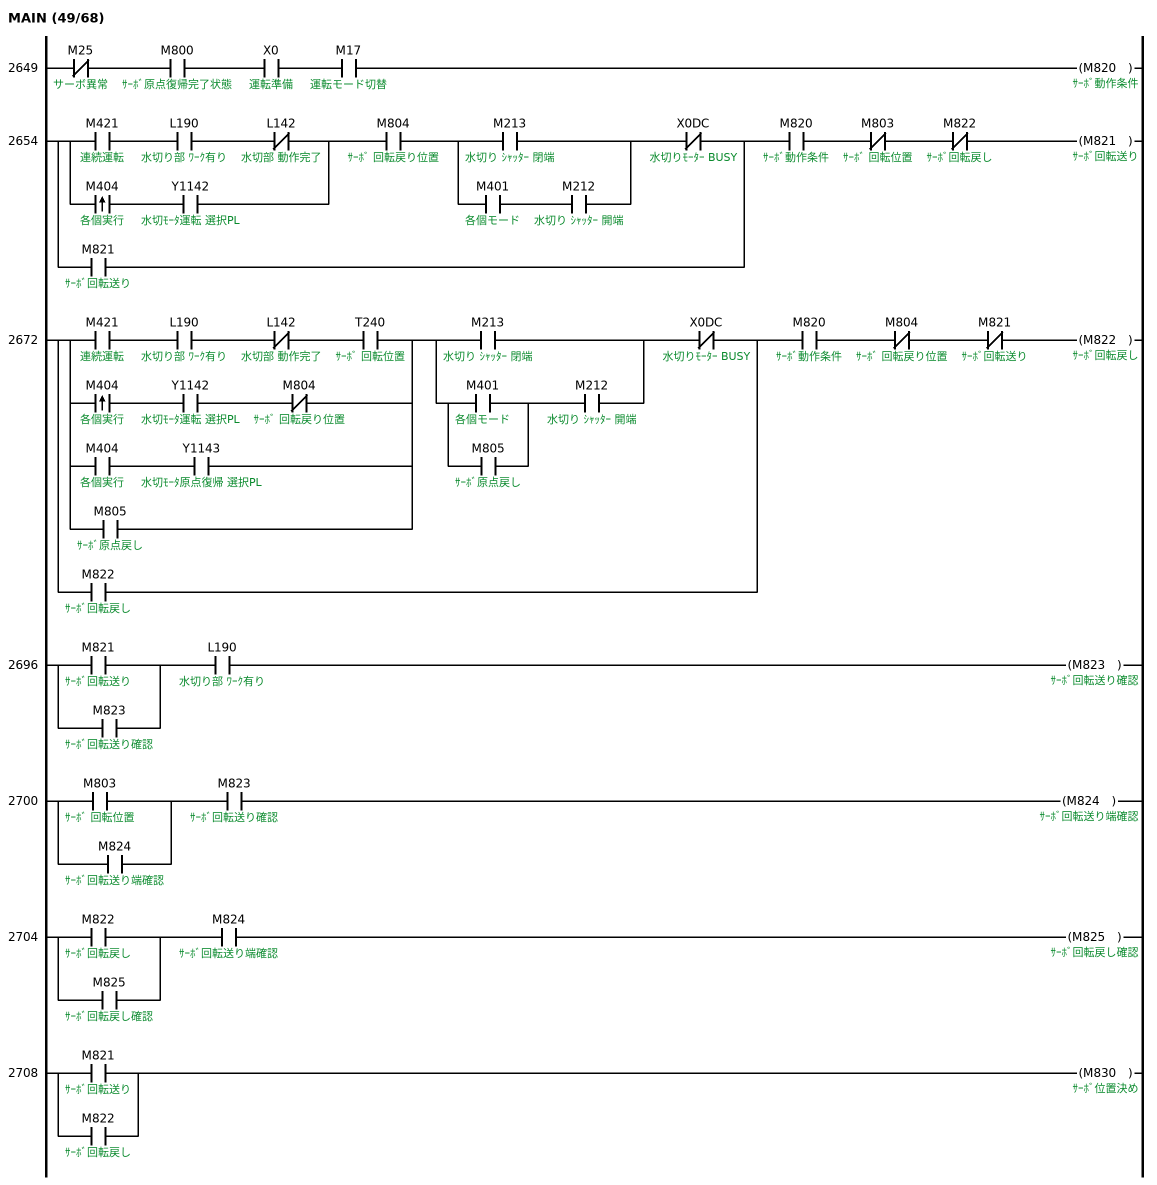
[picture p48: ladder of MAIN, rungs at steps 2649 to 2708]
2649  LDI     M25  ; サーボ異常
      AND     M800  ; ｻｰﾎﾞ原点復帰完了状態
      AND     X0  ; 運転準備
      AND     M17  ; 運転モード切替
      OUT     M820  ; ｻｰﾎﾞ動作条件
2654  LD      M421  ; 連続運転
      AND     L190  ; 水切り部 ﾜｰｸ有り
      ANI     L142  ; 水切部 動作完了
      LDP     M404  ; 各個実行
      AND     Y1142  ; 水切ﾓｰﾀ運転 選択PL
      ORB
      AND     M804  ; ｻｰﾎﾞ 回転戻り位置
      LD      M213  ; 水切り ｼｬｯﾀｰ 閉端
      LD      M401  ; 各個モード
      AND     M212  ; 水切り ｼｬｯﾀｰ 開端
      ORB
      ANB
      ANI     X0DC  ; 水切りﾓｰﾀｰ BUSY
      OR      M821  ; ｻｰﾎﾞ回転送り
      AND     M820  ; ｻｰﾎﾞ動作条件
      ANI     M803  ; ｻｰﾎﾞ 回転位置
      ANI     M822  ; ｻｰﾎﾞ回転戻し
      OUT     M821  ; ｻｰﾎﾞ回転送り
2672  LD      M421  ; 連続運転
      AND     L190  ; 水切り部 ﾜｰｸ有り
      ANI     L142  ; 水切部 動作完了
      AND     T240  ; ｻｰﾎﾞ 回転位置
      LDP     M404  ; 各個実行
      AND     Y1142  ; 水切ﾓｰﾀ運転 選択PL
      ANI     M804  ; ｻｰﾎﾞ 回転戻り位置
      ORB
      LD      M404  ; 各個実行
      AND     Y1143  ; 水切ﾓｰﾀ原点復帰 選択PL
      ORB
      OR      M805  ; ｻｰﾎﾞ原点戻し
      LD      M213  ; 水切り ｼｬｯﾀｰ 閉端
      LD      M401  ; 各個モード
      OR      M805  ; ｻｰﾎﾞ原点戻し
      AND     M212  ; 水切り ｼｬｯﾀｰ 開端
      ORB
      ANB
      ANI     X0DC  ; 水切りﾓｰﾀｰ BUSY
      OR      M822  ; ｻｰﾎﾞ回転戻し
      AND     M820  ; ｻｰﾎﾞ動作条件
      ANI     M804  ; ｻｰﾎﾞ 回転戻り位置
      ANI     M821  ; ｻｰﾎﾞ回転送り
      OUT     M822  ; ｻｰﾎﾞ回転戻し
2696  LD      M821  ; ｻｰﾎﾞ回転送り
      OR      M823  ; ｻｰﾎﾞ回転送り確認
      AND     L190  ; 水切り部 ﾜｰｸ有り
      OUT     M823  ; ｻｰﾎﾞ回転送り確認
2700  LD      M803  ; ｻｰﾎﾞ 回転位置
      OR      M824  ; ｻｰﾎﾞ回転送り端確認
      AND     M823  ; ｻｰﾎﾞ回転送り確認
      OUT     M824  ; ｻｰﾎﾞ回転送り端確認
2704  LD      M822  ; ｻｰﾎﾞ回転戻し
      OR      M825  ; ｻｰﾎﾞ回転戻し確認
      AND     M824  ; ｻｰﾎﾞ回転送り端確認
      OUT     M825  ; ｻｰﾎﾞ回転戻し確認
2708  LD      M821  ; ｻｰﾎﾞ回転送り
      OR      M822  ; ｻｰﾎﾞ回転戻し
      OUT     M830  ; ｻｰﾎﾞ位置決め
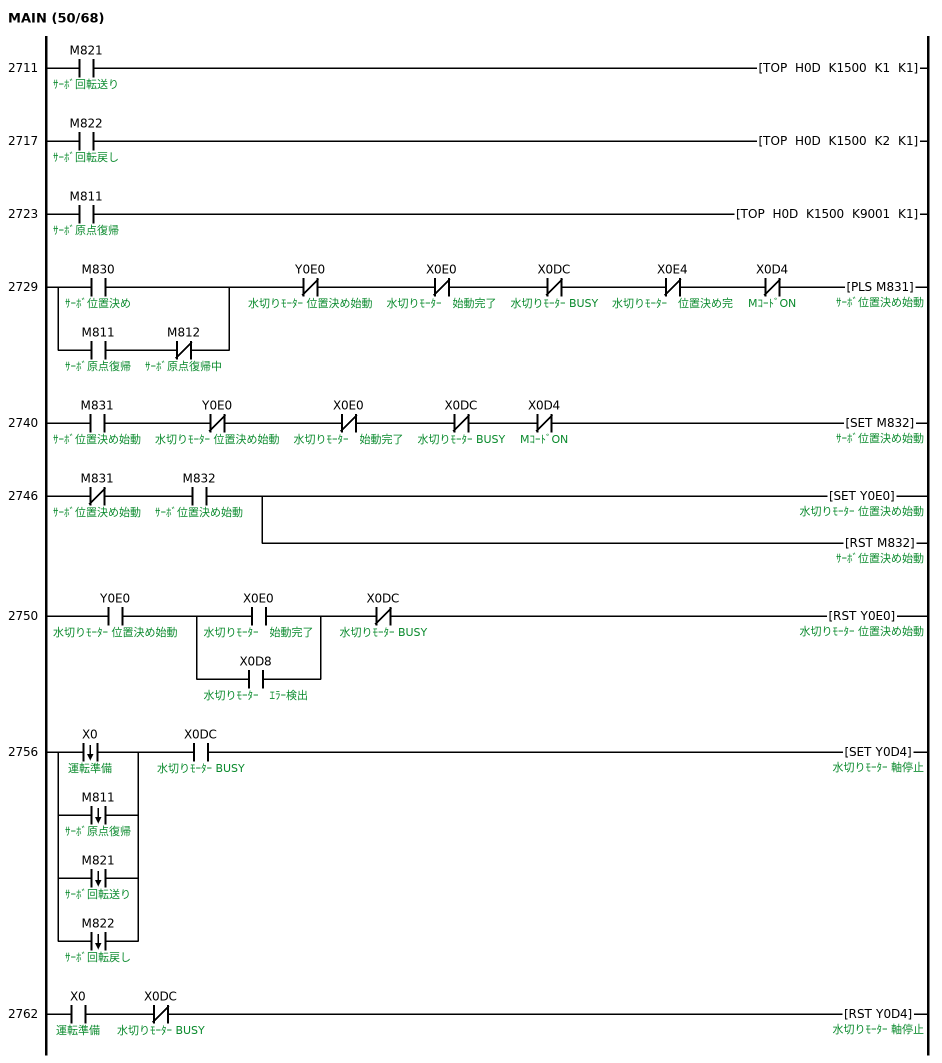
2711  LD      M821  ; ｻｰﾎﾞ回転送り
      TOP     H0D K1500 K1 K1
2717  LD      M822  ; ｻｰﾎﾞ回転戻し
      TOP     H0D K1500 K2 K1
2723  LD      M811  ; ｻｰﾎﾞ原点復帰
      TOP     H0D K1500 K9001 K1
2729  LD      M830  ; ｻｰﾎﾞ位置決め
      LD      M811  ; ｻｰﾎﾞ原点復帰
      ANI     M812  ; ｻｰﾎﾞ原点復帰中
      ORB
      ANI     Y0E0  ; 水切りﾓｰﾀｰ 位置決め始動
      ANI     X0E0  ; 水切りﾓｰﾀｰ　始動完了
      ANI     X0DC  ; 水切りﾓｰﾀｰ BUSY
      ANI     X0E4  ; 水切りﾓｰﾀｰ　位置決め完
      ANI     X0D4  ; MｺｰﾄﾞON
      PLS     M831  ; ｻｰﾎﾞ位置決め始動
2740  LD      M831  ; ｻｰﾎﾞ位置決め始動
      ANI     Y0E0  ; 水切りﾓｰﾀｰ 位置決め始動
      ANI     X0E0  ; 水切りﾓｰﾀｰ　始動完了
      ANI     X0DC  ; 水切りﾓｰﾀｰ BUSY
      ANI     X0D4  ; MｺｰﾄﾞON
      SET     M832  ; ｻｰﾎﾞ位置決め始動
2746  LDI     M831  ; ｻｰﾎﾞ位置決め始動
      AND     M832  ; ｻｰﾎﾞ位置決め始動
      SET     Y0E0  ; 水切りﾓｰﾀｰ 位置決め始動
      RST     M832  ; ｻｰﾎﾞ位置決め始動
2750  LD      Y0E0  ; 水切りﾓｰﾀｰ 位置決め始動
      LD      X0E0  ; 水切りﾓｰﾀｰ　始動完了
      OR      X0D8  ; 水切りﾓｰﾀｰ　ｴﾗｰ検出
      ANB
      ANI     X0DC  ; 水切りﾓｰﾀｰ BUSY
      RST     Y0E0  ; 水切りﾓｰﾀｰ 位置決め始動
2756  LDF     X0  ; 運転準備
      ORF     M811  ; ｻｰﾎﾞ原点復帰
      ORF     M821  ; ｻｰﾎﾞ回転送り
      ORF     M822  ; ｻｰﾎﾞ回転戻し
      AND     X0DC  ; 水切りﾓｰﾀｰ BUSY
      SET     Y0D4  ; 水切りﾓｰﾀｰ 軸停止
2762  LD      X0  ; 運転準備
      ANI     X0DC  ; 水切りﾓｰﾀｰ BUSY
      RST     Y0D4  ; 水切りﾓｰﾀｰ 軸停止
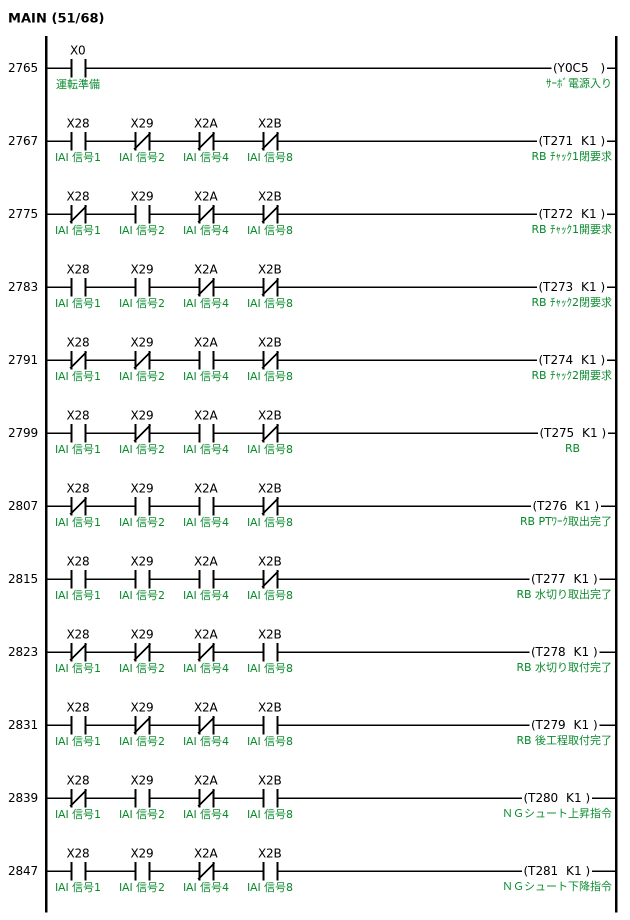
2765  LD      X0  ; 運転準備
      OUT     Y0C5  ; ｻｰﾎﾞ電源入り
2767  LD      X28  ; IAI 信号1
      ANI     X29  ; IAI 信号2
      ANI     X2A  ; IAI 信号4
      ANI     X2B  ; IAI 信号8
      OUT     T271 K1  ; RB ﾁｬｯｸ1閉要求
2775  LDI     X28  ; IAI 信号1
      AND     X29  ; IAI 信号2
      ANI     X2A  ; IAI 信号4
      ANI     X2B  ; IAI 信号8
      OUT     T272 K1  ; RB ﾁｬｯｸ1開要求
2783  LD      X28  ; IAI 信号1
      AND     X29  ; IAI 信号2
      ANI     X2A  ; IAI 信号4
      ANI     X2B  ; IAI 信号8
      OUT     T273 K1  ; RB ﾁｬｯｸ2閉要求
2791  LDI     X28  ; IAI 信号1
      ANI     X29  ; IAI 信号2
      AND     X2A  ; IAI 信号4
      ANI     X2B  ; IAI 信号8
      OUT     T274 K1  ; RB ﾁｬｯｸ2開要求
2799  LD      X28  ; IAI 信号1
      ANI     X29  ; IAI 信号2
      AND     X2A  ; IAI 信号4
      ANI     X2B  ; IAI 信号8
      OUT     T275 K1  ; RB
2807  LDI     X28  ; IAI 信号1
      AND     X29  ; IAI 信号2
      AND     X2A  ; IAI 信号4
      ANI     X2B  ; IAI 信号8
      OUT     T276 K1  ; RB PTﾜｰｸ取出完了
2815  LD      X28  ; IAI 信号1
      AND     X29  ; IAI 信号2
      AND     X2A  ; IAI 信号4
      ANI     X2B  ; IAI 信号8
      OUT     T277 K1  ; RB 水切り取出完了
2823  LDI     X28  ; IAI 信号1
      ANI     X29  ; IAI 信号2
      ANI     X2A  ; IAI 信号4
      AND     X2B  ; IAI 信号8
      OUT     T278 K1  ; RB 水切り取付完了
2831  LD      X28  ; IAI 信号1
      ANI     X29  ; IAI 信号2
      ANI     X2A  ; IAI 信号4
      AND     X2B  ; IAI 信号8
      OUT     T279 K1  ; RB 後工程取付完了
2839  LDI     X28  ; IAI 信号1
      AND     X29  ; IAI 信号2
      ANI     X2A  ; IAI 信号4
      AND     X2B  ; IAI 信号8
      OUT     T280 K1  ; ＮＧシュート上昇指令
2847  LD      X28  ; IAI 信号1
      AND     X29  ; IAI 信号2
      ANI     X2A  ; IAI 信号4
      AND     X2B  ; IAI 信号8
      OUT     T281 K1  ; ＮＧシュート下降指令
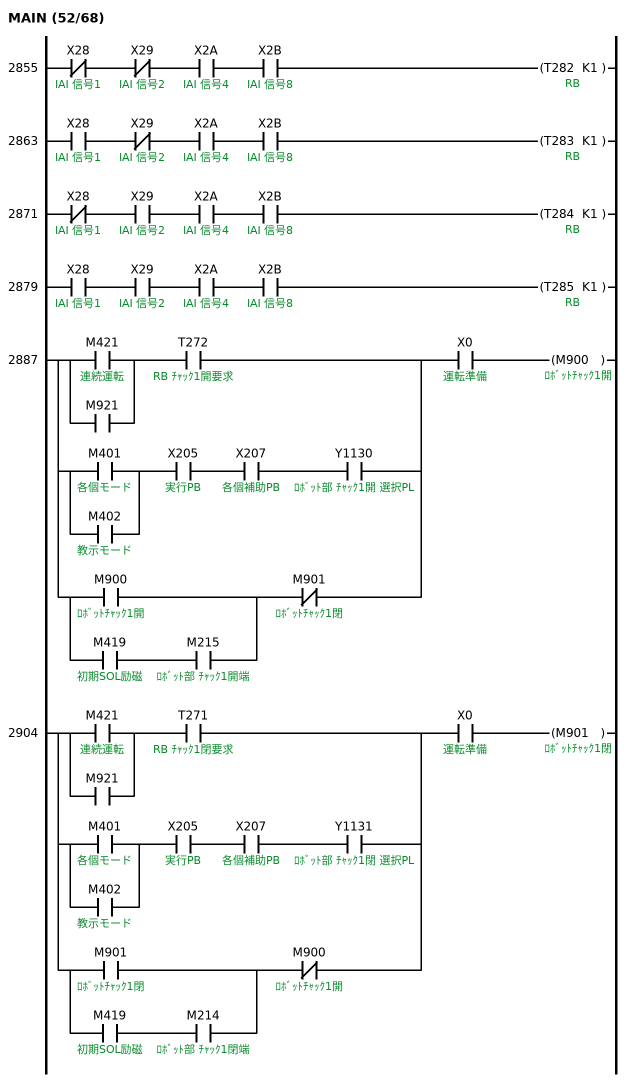
2855  LDI     X28  ; IAI 信号1
      ANI     X29  ; IAI 信号2
      AND     X2A  ; IAI 信号4
      AND     X2B  ; IAI 信号8
      OUT     T282 K1  ; RB
2863  LD      X28  ; IAI 信号1
      ANI     X29  ; IAI 信号2
      AND     X2A  ; IAI 信号4
      AND     X2B  ; IAI 信号8
      OUT     T283 K1  ; RB
2871  LDI     X28  ; IAI 信号1
      AND     X29  ; IAI 信号2
      AND     X2A  ; IAI 信号4
      AND     X2B  ; IAI 信号8
      OUT     T284 K1  ; RB
2879  LD      X28  ; IAI 信号1
      AND     X29  ; IAI 信号2
      AND     X2A  ; IAI 信号4
      AND     X2B  ; IAI 信号8
      OUT     T285 K1  ; RB
2887  LD      M421  ; 連続運転
      OR      M921
      AND     T272  ; RB ﾁｬｯｸ1開要求
      LD      M401  ; 各個モード
      OR      M402  ; 教示モード
      AND     X205  ; 実行PB
      AND     X207  ; 各個補助PB
      AND     Y1130  ; ﾛﾎﾞｯﾄ部 ﾁｬｯｸ1開 選択PL
      ORB
      LD      M900  ; ﾛﾎﾞｯﾄﾁｬｯｸ1開
      LD      M419  ; 初期SOL励磁
      AND     M215  ; ﾛﾎﾞｯﾄ部 ﾁｬｯｸ1開端
      ORB
      ANI     M901  ; ﾛﾎﾞｯﾄﾁｬｯｸ1閉
      ORB
      AND     X0  ; 運転準備
      OUT     M900  ; ﾛﾎﾞｯﾄﾁｬｯｸ1開
2904  LD      M421  ; 連続運転
      OR      M921
      AND     T271  ; RB ﾁｬｯｸ1閉要求
      LD      M401  ; 各個モード
      OR      M402  ; 教示モード
      AND     X205  ; 実行PB
      AND     X207  ; 各個補助PB
      AND     Y1131  ; ﾛﾎﾞｯﾄ部 ﾁｬｯｸ1閉 選択PL
      ORB
      LD      M901  ; ﾛﾎﾞｯﾄﾁｬｯｸ1閉
      LD      M419  ; 初期SOL励磁
      AND     M214  ; ﾛﾎﾞｯﾄ部 ﾁｬｯｸ1閉端
      ORB
      ANI     M900  ; ﾛﾎﾞｯﾄﾁｬｯｸ1開
      ORB
      AND     X0  ; 運転準備
      OUT     M901  ; ﾛﾎﾞｯﾄﾁｬｯｸ1閉
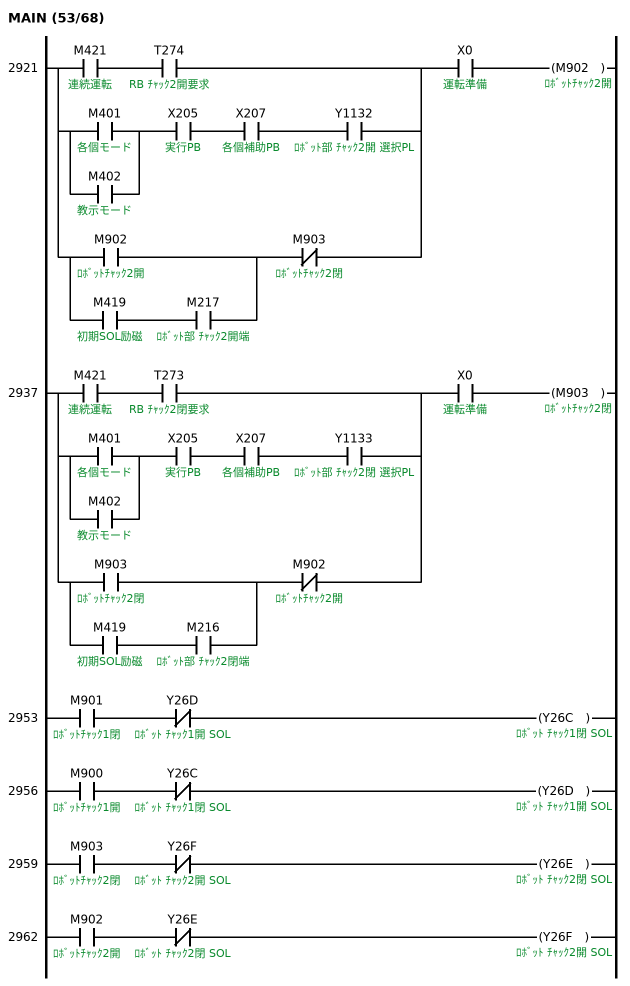
2921  LD      M421  ; 連続運転
      AND     T274  ; RB ﾁｬｯｸ2開要求
      LD      M401  ; 各個モード
      OR      M402  ; 教示モード
      AND     X205  ; 実行PB
      AND     X207  ; 各個補助PB
      AND     Y1132  ; ﾛﾎﾞｯﾄ部 ﾁｬｯｸ2開 選択PL
      ORB
      LD      M902  ; ﾛﾎﾞｯﾄﾁｬｯｸ2開
      LD      M419  ; 初期SOL励磁
      AND     M217  ; ﾛﾎﾞｯﾄ部 ﾁｬｯｸ2開端
      ORB
      ANI     M903  ; ﾛﾎﾞｯﾄﾁｬｯｸ2閉
      ORB
      AND     X0  ; 運転準備
      OUT     M902  ; ﾛﾎﾞｯﾄﾁｬｯｸ2開
2937  LD      M421  ; 連続運転
      AND     T273  ; RB ﾁｬｯｸ2閉要求
      LD      M401  ; 各個モード
      OR      M402  ; 教示モード
      AND     X205  ; 実行PB
      AND     X207  ; 各個補助PB
      AND     Y1133  ; ﾛﾎﾞｯﾄ部 ﾁｬｯｸ2閉 選択PL
      ORB
      LD      M903  ; ﾛﾎﾞｯﾄﾁｬｯｸ2閉
      LD      M419  ; 初期SOL励磁
      AND     M216  ; ﾛﾎﾞｯﾄ部 ﾁｬｯｸ2閉端
      ORB
      ANI     M902  ; ﾛﾎﾞｯﾄﾁｬｯｸ2開
      ORB
      AND     X0  ; 運転準備
      OUT     M903  ; ﾛﾎﾞｯﾄﾁｬｯｸ2閉
2953  LD      M901  ; ﾛﾎﾞｯﾄﾁｬｯｸ1閉
      ANI     Y26D  ; ﾛﾎﾞｯﾄ ﾁｬｯｸ1開 SOL
      OUT     Y26C  ; ﾛﾎﾞｯﾄ ﾁｬｯｸ1閉 SOL
2956  LD      M900  ; ﾛﾎﾞｯﾄﾁｬｯｸ1開
      ANI     Y26C  ; ﾛﾎﾞｯﾄ ﾁｬｯｸ1閉 SOL
      OUT     Y26D  ; ﾛﾎﾞｯﾄ ﾁｬｯｸ1開 SOL
2959  LD      M903  ; ﾛﾎﾞｯﾄﾁｬｯｸ2閉
      ANI     Y26F  ; ﾛﾎﾞｯﾄ ﾁｬｯｸ2開 SOL
      OUT     Y26E  ; ﾛﾎﾞｯﾄ ﾁｬｯｸ2閉 SOL
2962  LD      M902  ; ﾛﾎﾞｯﾄﾁｬｯｸ2開
      ANI     Y26E  ; ﾛﾎﾞｯﾄ ﾁｬｯｸ2閉 SOL
      OUT     Y26F  ; ﾛﾎﾞｯﾄ ﾁｬｯｸ2開 SOL
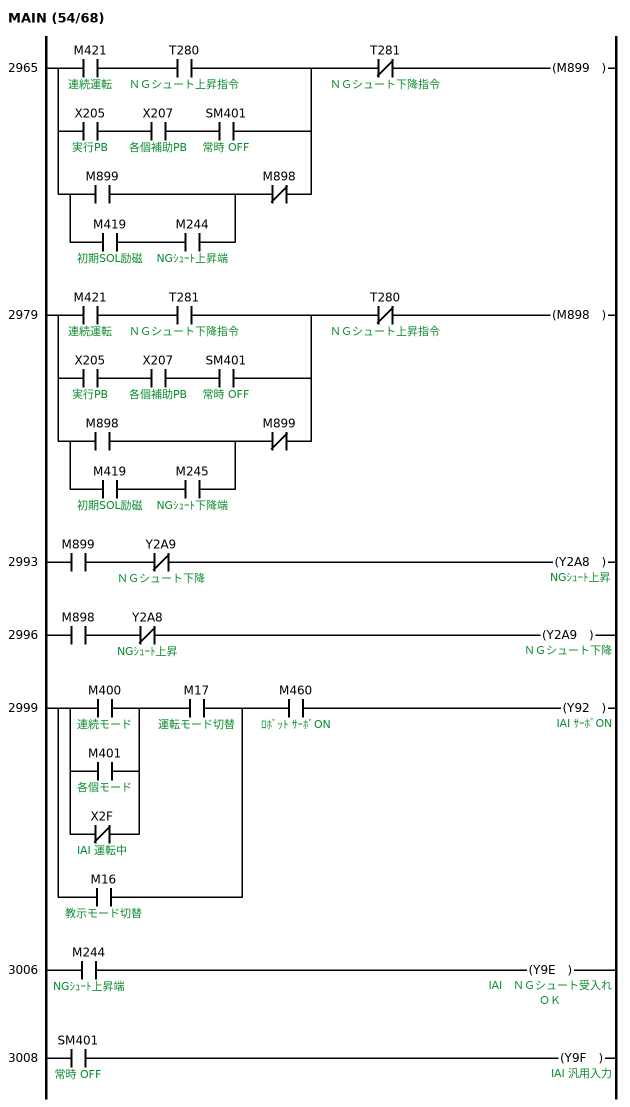
2965  LD      M421  ; 連続運転
      AND     T280  ; ＮＧシュート上昇指令
      LD      X205  ; 実行PB
      AND     X207  ; 各個補助PB
      AND     SM401  ; 常時 OFF
      ORB
      LD      M899
      LD      M419  ; 初期SOL励磁
      AND     M244  ; NGｼｭｰﾄ上昇端
      ORB
      ANI     M898
      ORB
      ANI     T281  ; ＮＧシュート下降指令
      OUT     M899
2979  LD      M421  ; 連続運転
      AND     T281  ; ＮＧシュート下降指令
      LD      X205  ; 実行PB
      AND     X207  ; 各個補助PB
      AND     SM401  ; 常時 OFF
      ORB
      LD      M898
      LD      M419  ; 初期SOL励磁
      AND     M245  ; NGｼｭｰﾄ下降端
      ORB
      ANI     M899
      ORB
      ANI     T280  ; ＮＧシュート上昇指令
      OUT     M898
2993  LD      M899
      ANI     Y2A9  ; ＮＧシュート下降
      OUT     Y2A8  ; NGｼｭｰﾄ上昇
2996  LD      M898
      ANI     Y2A8  ; NGｼｭｰﾄ上昇
      OUT     Y2A9  ; ＮＧシュート下降
2999  LD      M400  ; 連続モード
      OR      M401  ; 各個モード
      ORI     X2F  ; IAI 運転中
      AND     M17  ; 運転モード切替
      OR      M16  ; 教示モード切替
      AND     M460  ; ﾛﾎﾞｯﾄ ｻｰﾎﾞON
      OUT     Y92  ; IAI ｻｰﾎﾞON
3006  LD      M244  ; NGｼｭｰﾄ上昇端
      OUT     Y9E  ; IAI　ＮＧシュート受入れＯＫ
3008  LD      SM401  ; 常時 OFF
      OUT     Y9F  ; IAI 汎用入力
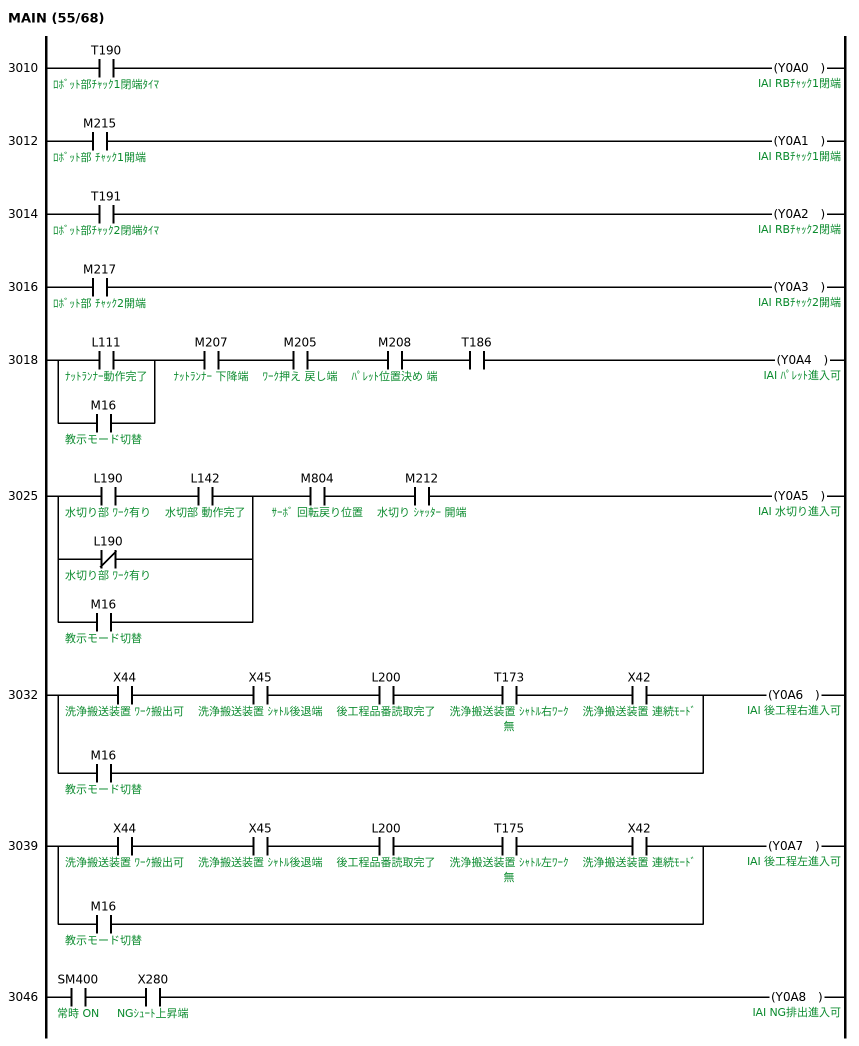
3010  LD      T190  ; ﾛﾎﾞｯﾄ部ﾁｬｯｸ1閉端ﾀｲﾏ
      OUT     Y0A0  ; IAI RBﾁｬｯｸ1閉端
3012  LD      M215  ; ﾛﾎﾞｯﾄ部 ﾁｬｯｸ1開端
      OUT     Y0A1  ; IAI RBﾁｬｯｸ1開端
3014  LD      T191  ; ﾛﾎﾞｯﾄ部ﾁｬｯｸ2閉端ﾀｲﾏ
      OUT     Y0A2  ; IAI RBﾁｬｯｸ2閉端
3016  LD      M217  ; ﾛﾎﾞｯﾄ部 ﾁｬｯｸ2開端
      OUT     Y0A3  ; IAI RBﾁｬｯｸ2開端
3018  LD      L111  ; ﾅｯﾄﾗﾝﾅｰ動作完了
      OR      M16  ; 教示モード切替
      AND     M207  ; ﾅｯﾄﾗﾝﾅｰ 下降端
      AND     M205  ; ﾜｰｸ押え 戻し端
      AND     M208  ; ﾊﾟﾚｯﾄ位置決め 端
      AND     T186
      OUT     Y0A4  ; IAI ﾊﾟﾚｯﾄ進入可
3025  LD      L190  ; 水切り部 ﾜｰｸ有り
      AND     L142  ; 水切部 動作完了
      ORI     L190  ; 水切り部 ﾜｰｸ有り
      OR      M16  ; 教示モード切替
      AND     M804  ; ｻｰﾎﾞ 回転戻り位置
      AND     M212  ; 水切り ｼｬｯﾀｰ 開端
      OUT     Y0A5  ; IAI 水切り進入可
3032  LD      X44  ; 洗浄搬送装置 ﾜｰｸ搬出可
      AND     X45  ; 洗浄搬送装置 ｼｬﾄﾙ後退端
      AND     L200  ; 後工程品番読取完了
      AND     T173  ; 洗浄搬送装置 ｼｬﾄﾙ右ﾜｰｸ無
      AND     X42  ; 洗浄搬送装置 連続ﾓｰﾄﾞ
      OR      M16  ; 教示モード切替
      OUT     Y0A6  ; IAI 後工程右進入可
3039  LD      X44  ; 洗浄搬送装置 ﾜｰｸ搬出可
      AND     X45  ; 洗浄搬送装置 ｼｬﾄﾙ後退端
      AND     L200  ; 後工程品番読取完了
      AND     T175  ; 洗浄搬送装置 ｼｬﾄﾙ左ﾜｰｸ無
      AND     X42  ; 洗浄搬送装置 連続ﾓｰﾄﾞ
      OR      M16  ; 教示モード切替
      OUT     Y0A7  ; IAI 後工程左進入可
3046  LD      SM400  ; 常時 ON
      AND     X280  ; NGｼｭｰﾄ上昇端
      OUT     Y0A8  ; IAI NG排出進入可
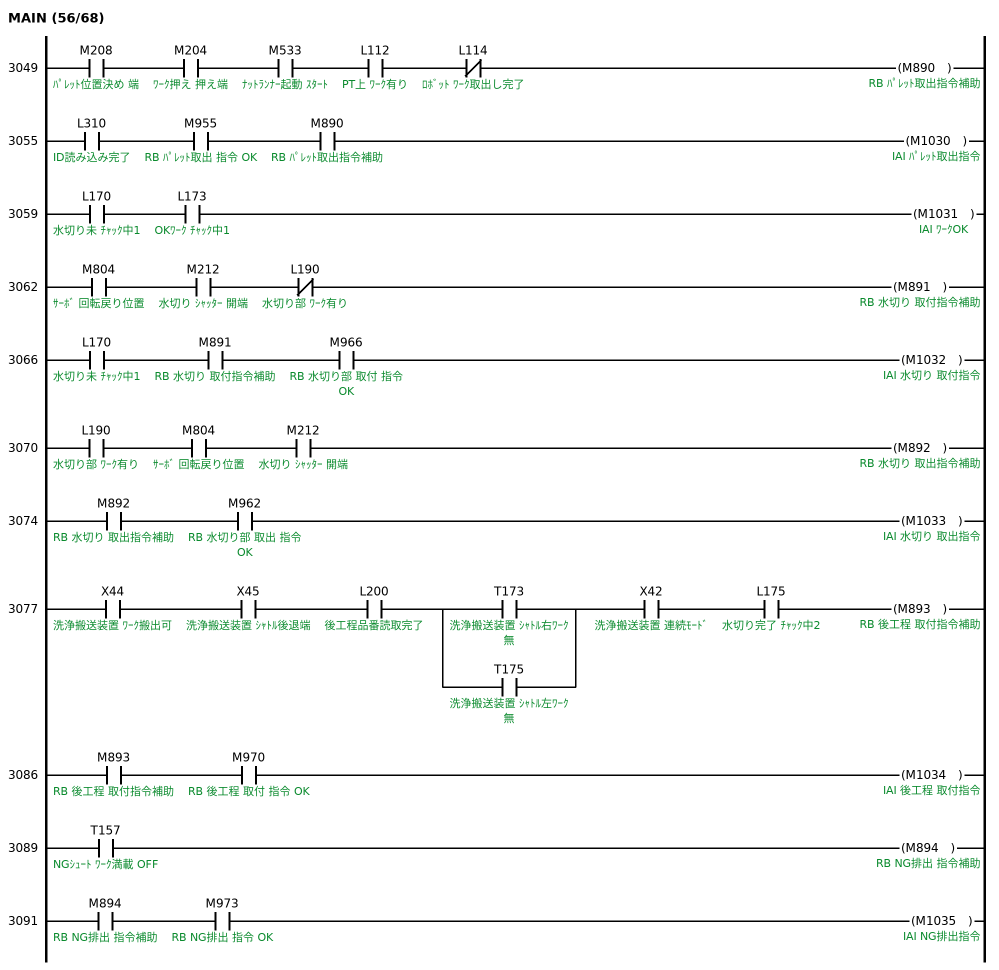
3049  LD      M208  ; ﾊﾟﾚｯﾄ位置決め 端
      AND     M204  ; ﾜｰｸ押え 押え端
      AND     M533  ; ﾅｯﾄﾗﾝﾅｰ起動 ｽﾀｰﾄ
      AND     L112  ; PT上 ﾜｰｸ有り
      ANI     L114  ; ﾛﾎﾞｯﾄ ﾜｰｸ取出し完了
      OUT     M890  ; RB ﾊﾟﾚｯﾄ取出指令補助
3055  LD      L310  ; ID読み込み完了
      AND     M955  ; RB ﾊﾟﾚｯﾄ取出 指令 OK
      AND     M890  ; RB ﾊﾟﾚｯﾄ取出指令補助
      OUT     M1030  ; IAI ﾊﾟﾚｯﾄ取出指令
3059  LD      L170  ; 水切り未 ﾁｬｯｸ中1
      AND     L173  ; OKﾜｰｸ ﾁｬｯｸ中1
      OUT     M1031  ; IAI ﾜｰｸOK
3062  LD      M804  ; ｻｰﾎﾞ 回転戻り位置
      AND     M212  ; 水切り ｼｬｯﾀｰ 開端
      ANI     L190  ; 水切り部 ﾜｰｸ有り
      OUT     M891  ; RB 水切り 取付指令補助
3066  LD      L170  ; 水切り未 ﾁｬｯｸ中1
      AND     M891  ; RB 水切り 取付指令補助
      AND     M966  ; RB 水切り部 取付 指令 OK
      OUT     M1032  ; IAI 水切り 取付指令
3070  LD      L190  ; 水切り部 ﾜｰｸ有り
      AND     M804  ; ｻｰﾎﾞ 回転戻り位置
      AND     M212  ; 水切り ｼｬｯﾀｰ 開端
      OUT     M892  ; RB 水切り 取出指令補助
3074  LD      M892  ; RB 水切り 取出指令補助
      AND     M962  ; RB 水切り部 取出 指令 OK
      OUT     M1033  ; IAI 水切り 取出指令
3077  LD      X44  ; 洗浄搬送装置 ﾜｰｸ搬出可
      AND     X45  ; 洗浄搬送装置 ｼｬﾄﾙ後退端
      AND     L200  ; 後工程品番読取完了
      LD      T173  ; 洗浄搬送装置 ｼｬﾄﾙ右ﾜｰｸ無
      OR      T175  ; 洗浄搬送装置 ｼｬﾄﾙ左ﾜｰｸ無
      ANB
      AND     X42  ; 洗浄搬送装置 連続ﾓｰﾄﾞ
      AND     L175  ; 水切り完了 ﾁｬｯｸ中2
      OUT     M893  ; RB 後工程 取付指令補助
3086  LD      M893  ; RB 後工程 取付指令補助
      AND     M970  ; RB 後工程 取付 指令 OK
      OUT     M1034  ; IAI 後工程 取付指令
3089  LD      T157  ; NGｼｭｰﾄ ﾜｰｸ満載 OFF
      OUT     M894  ; RB NG排出 指令補助
3091  LD      M894  ; RB NG排出 指令補助
      AND     M973  ; RB NG排出 指令 OK
      OUT     M1035  ; IAI NG排出指令
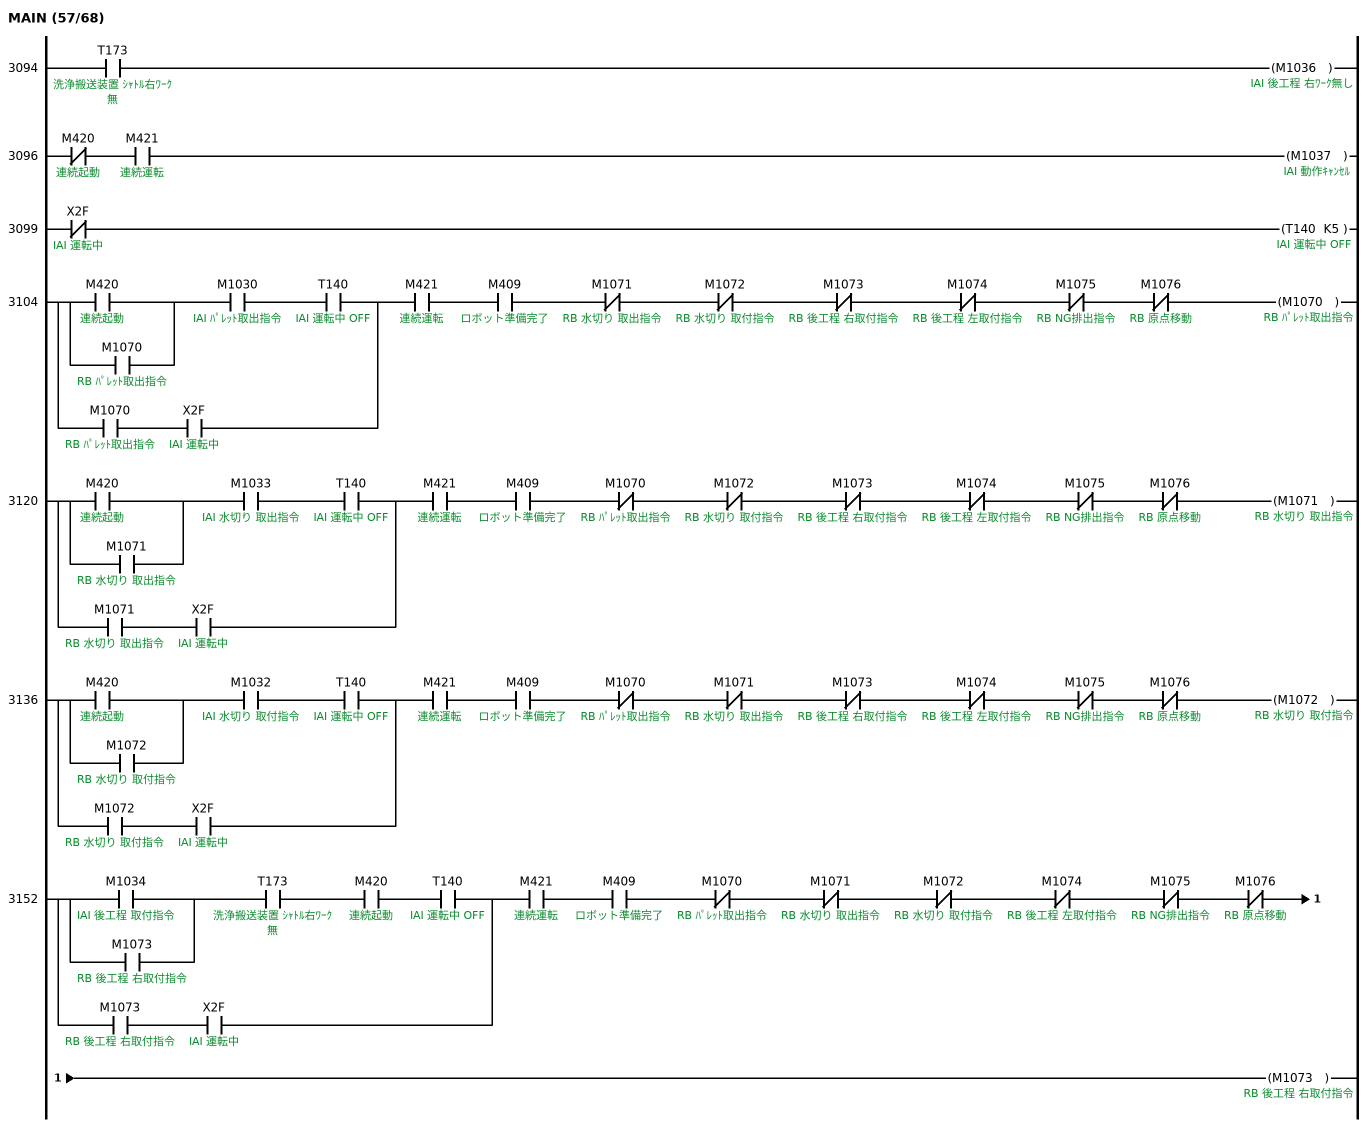
3094  LD      T173  ; 洗浄搬送装置 ｼｬﾄﾙ右ﾜｰｸ無
      OUT     M1036  ; IAI 後工程 右ﾜｰｸ無し
3096  LDI     M420  ; 連続起動
      AND     M421  ; 連続運転
      OUT     M1037  ; IAI 動作ｷｬﾝｾﾙ
3099  LDI     X2F  ; IAI 運転中
      OUT     T140 K5  ; IAI 運転中 OFF
3104  LD      M420  ; 連続起動
      OR      M1070  ; RB ﾊﾟﾚｯﾄ取出指令
      AND     M1030  ; IAI ﾊﾟﾚｯﾄ取出指令
      AND     T140  ; IAI 運転中 OFF
      LD      M1070  ; RB ﾊﾟﾚｯﾄ取出指令
      AND     X2F  ; IAI 運転中
      ORB
      AND     M421  ; 連続運転
      AND     M409  ; ロボット準備完了
      ANI     M1071  ; RB 水切り 取出指令
      ANI     M1072  ; RB 水切り 取付指令
      ANI     M1073  ; RB 後工程 右取付指令
      ANI     M1074  ; RB 後工程 左取付指令
      ANI     M1075  ; RB NG排出指令
      ANI     M1076  ; RB 原点移動
      OUT     M1070  ; RB ﾊﾟﾚｯﾄ取出指令
3120  LD      M420  ; 連続起動
      OR      M1071  ; RB 水切り 取出指令
      AND     M1033  ; IAI 水切り 取出指令
      AND     T140  ; IAI 運転中 OFF
      LD      M1071  ; RB 水切り 取出指令
      AND     X2F  ; IAI 運転中
      ORB
      AND     M421  ; 連続運転
      AND     M409  ; ロボット準備完了
      ANI     M1070  ; RB ﾊﾟﾚｯﾄ取出指令
      ANI     M1072  ; RB 水切り 取付指令
      ANI     M1073  ; RB 後工程 右取付指令
      ANI     M1074  ; RB 後工程 左取付指令
      ANI     M1075  ; RB NG排出指令
      ANI     M1076  ; RB 原点移動
      OUT     M1071  ; RB 水切り 取出指令
3136  LD      M420  ; 連続起動
      OR      M1072  ; RB 水切り 取付指令
      AND     M1032  ; IAI 水切り 取付指令
      AND     T140  ; IAI 運転中 OFF
      LD      M1072  ; RB 水切り 取付指令
      AND     X2F  ; IAI 運転中
      ORB
      AND     M421  ; 連続運転
      AND     M409  ; ロボット準備完了
      ANI     M1070  ; RB ﾊﾟﾚｯﾄ取出指令
      ANI     M1071  ; RB 水切り 取出指令
      ANI     M1073  ; RB 後工程 右取付指令
      ANI     M1074  ; RB 後工程 左取付指令
      ANI     M1075  ; RB NG排出指令
      ANI     M1076  ; RB 原点移動
      OUT     M1072  ; RB 水切り 取付指令
3152  LD      M1034  ; IAI 後工程 取付指令
      OR      M1073  ; RB 後工程 右取付指令
      AND     T173  ; 洗浄搬送装置 ｼｬﾄﾙ右ﾜｰｸ無
      AND     M420  ; 連続起動
      AND     T140  ; IAI 運転中 OFF
      LD      M1073  ; RB 後工程 右取付指令
      AND     X2F  ; IAI 運転中
      ORB
      AND     M421  ; 連続運転
      AND     M409  ; ロボット準備完了
      ANI     M1070  ; RB ﾊﾟﾚｯﾄ取出指令
      ANI     M1071  ; RB 水切り 取出指令
      ANI     M1072  ; RB 水切り 取付指令
      ANI     M1074  ; RB 後工程 左取付指令
      ANI     M1075  ; RB NG排出指令
      ANI     M1076  ; RB 原点移動
      OUT     M1073  ; RB 後工程 右取付指令
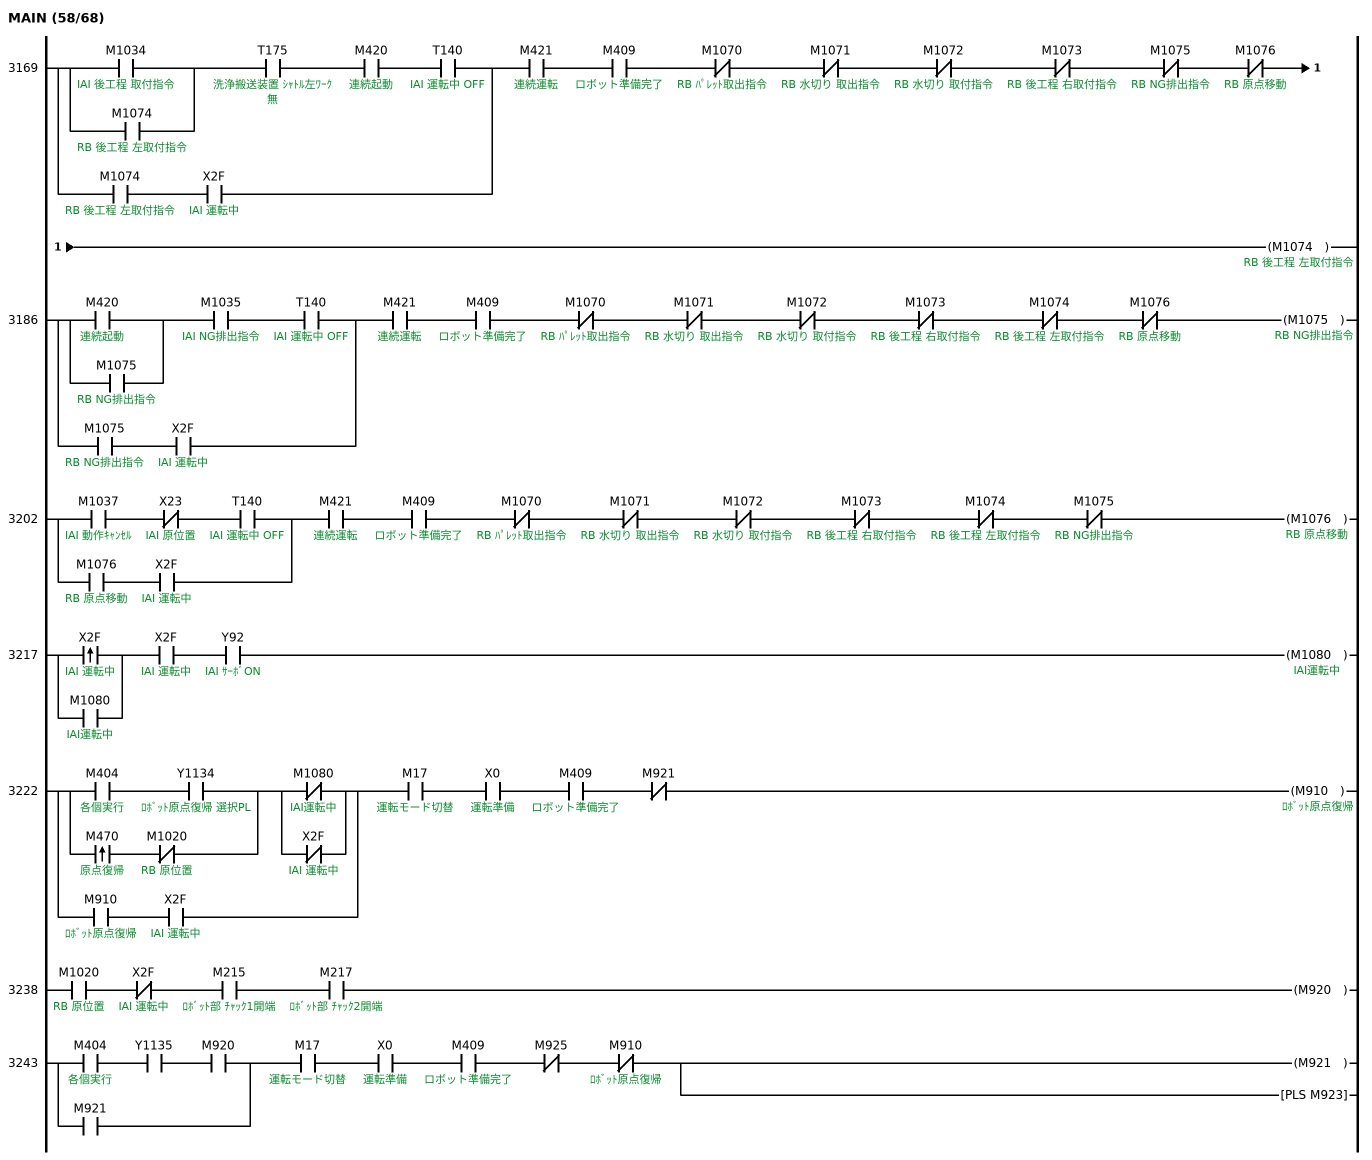
3169  LD      M1034  ; IAI 後工程 取付指令
      OR      M1074  ; RB 後工程 左取付指令
      AND     T175  ; 洗浄搬送装置 ｼｬﾄﾙ左ﾜｰｸ無
      AND     M420  ; 連続起動
      AND     T140  ; IAI 運転中 OFF
      LD      M1074  ; RB 後工程 左取付指令
      AND     X2F  ; IAI 運転中
      ORB
      AND     M421  ; 連続運転
      AND     M409  ; ロボット準備完了
      ANI     M1070  ; RB ﾊﾟﾚｯﾄ取出指令
      ANI     M1071  ; RB 水切り 取出指令
      ANI     M1072  ; RB 水切り 取付指令
      ANI     M1073  ; RB 後工程 右取付指令
      ANI     M1075  ; RB NG排出指令
      ANI     M1076  ; RB 原点移動
      OUT     M1074  ; RB 後工程 左取付指令
3186  LD      M420  ; 連続起動
      OR      M1075  ; RB NG排出指令
      AND     M1035  ; IAI NG排出指令
      AND     T140  ; IAI 運転中 OFF
      LD      M1075  ; RB NG排出指令
      AND     X2F  ; IAI 運転中
      ORB
      AND     M421  ; 連続運転
      AND     M409  ; ロボット準備完了
      ANI     M1070  ; RB ﾊﾟﾚｯﾄ取出指令
      ANI     M1071  ; RB 水切り 取出指令
      ANI     M1072  ; RB 水切り 取付指令
      ANI     M1073  ; RB 後工程 右取付指令
      ANI     M1074  ; RB 後工程 左取付指令
      ANI     M1076  ; RB 原点移動
      OUT     M1075  ; RB NG排出指令
3202  LD      M1037  ; IAI 動作ｷｬﾝｾﾙ
      ANI     X23  ; IAI 原位置
      AND     T140  ; IAI 運転中 OFF
      LD      M1076  ; RB 原点移動
      AND     X2F  ; IAI 運転中
      ORB
      AND     M421  ; 連続運転
      AND     M409  ; ロボット準備完了
      ANI     M1070  ; RB ﾊﾟﾚｯﾄ取出指令
      ANI     M1071  ; RB 水切り 取出指令
      ANI     M1072  ; RB 水切り 取付指令
      ANI     M1073  ; RB 後工程 右取付指令
      ANI     M1074  ; RB 後工程 左取付指令
      ANI     M1075  ; RB NG排出指令
      OUT     M1076  ; RB 原点移動
3217  LDP     X2F  ; IAI 運転中
      OR      M1080  ; IAI運転中
      AND     X2F  ; IAI 運転中
      AND     Y92  ; IAI ｻｰﾎﾞON
      OUT     M1080  ; IAI運転中
3222  LD      M404  ; 各個実行
      AND     Y1134  ; ﾛﾎﾞｯﾄ原点復帰 選択PL
      LDP     M470  ; 原点復帰
      ANI     M1020  ; RB 原位置
      ORB
      LDI     M1080  ; IAI運転中
      ORI     X2F  ; IAI 運転中
      ANB
      LD      M910  ; ﾛﾎﾞｯﾄ原点復帰
      AND     X2F  ; IAI 運転中
      ORB
      AND     M17  ; 運転モード切替
      AND     X0  ; 運転準備
      AND     M409  ; ロボット準備完了
      ANI     M921
      OUT     M910  ; ﾛﾎﾞｯﾄ原点復帰
3238  LD      M1020  ; RB 原位置
      ANI     X2F  ; IAI 運転中
      AND     M215  ; ﾛﾎﾞｯﾄ部 ﾁｬｯｸ1開端
      AND     M217  ; ﾛﾎﾞｯﾄ部 ﾁｬｯｸ2開端
      OUT     M920
3243  LD      M404  ; 各個実行
      AND     Y1135
      AND     M920
      OR      M921
      AND     M17  ; 運転モード切替
      AND     X0  ; 運転準備
      AND     M409  ; ロボット準備完了
      ANI     M925
      ANI     M910  ; ﾛﾎﾞｯﾄ原点復帰
      OUT     M921
      PLS     M923
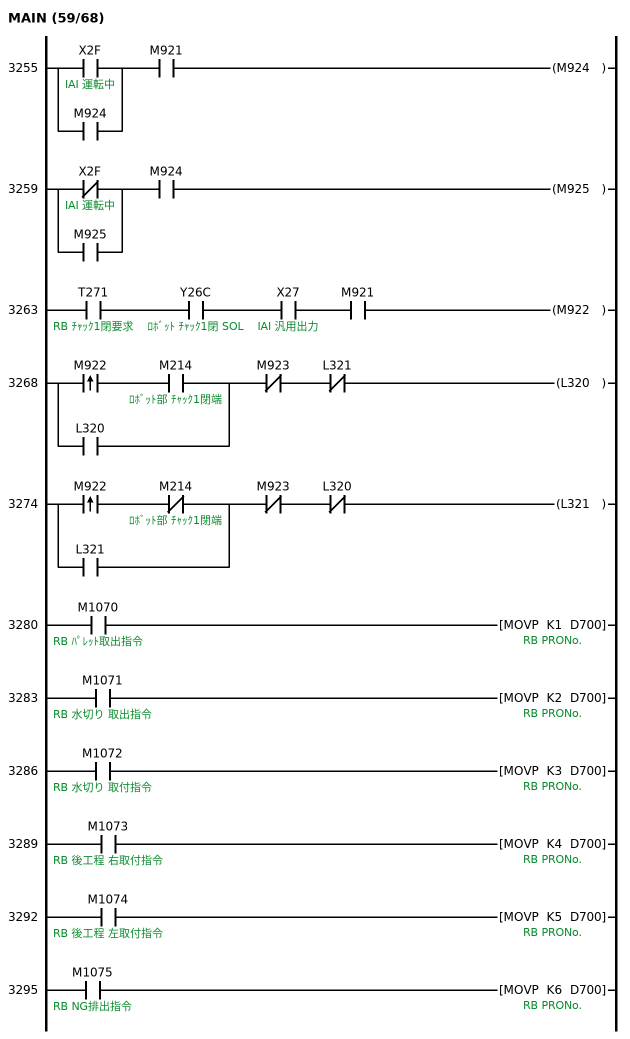
3255  LD      X2F  ; IAI 運転中
      OR      M924
      AND     M921
      OUT     M924
3259  LDI     X2F  ; IAI 運転中
      OR      M925
      AND     M924
      OUT     M925
3263  LD      T271  ; RB ﾁｬｯｸ1閉要求
      AND     Y26C  ; ﾛﾎﾞｯﾄ ﾁｬｯｸ1閉 SOL
      AND     X27  ; IAI 汎用出力
      AND     M921
      OUT     M922
3268  LDP     M922
      AND     M214  ; ﾛﾎﾞｯﾄ部 ﾁｬｯｸ1閉端
      OR      L320
      ANI     M923
      ANI     L321
      OUT     L320
3274  LDP     M922
      ANI     M214  ; ﾛﾎﾞｯﾄ部 ﾁｬｯｸ1閉端
      OR      L321
      ANI     M923
      ANI     L320
      OUT     L321
3280  LD      M1070  ; RB ﾊﾟﾚｯﾄ取出指令
      MOVP    K1 D700  ; RB PRONo.
3283  LD      M1071  ; RB 水切り 取出指令
      MOVP    K2 D700
3286  LD      M1072  ; RB 水切り 取付指令
      MOVP    K3 D700
3289  LD      M1073  ; RB 後工程 右取付指令
      MOVP    K4 D700
3292  LD      M1074  ; RB 後工程 左取付指令
      MOVP    K5 D700
3295  LD      M1075  ; RB NG排出指令
      MOVP    K6 D700
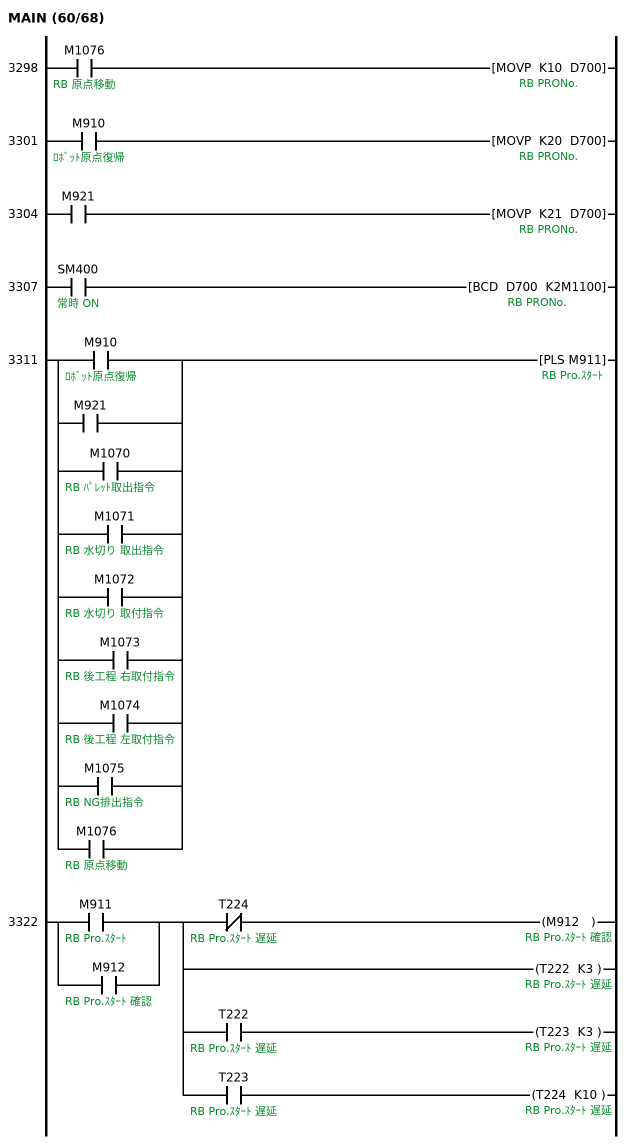
3298  LD      M1076  ; RB 原点移動
      MOVP    K10 D700
3301  LD      M910  ; ﾛﾎﾞｯﾄ原点復帰
      MOVP    K20 D700
3304  LD      M921
      MOVP    K21 D700
3307  LD      SM400  ; 常時 ON
      BCD     D700 K2M1100  ; RB PRO No.1
3311  LD      M910  ; ﾛﾎﾞｯﾄ原点復帰
      OR      M921
      OR      M1070  ; RB ﾊﾟﾚｯﾄ取出指令
      OR      M1071  ; RB 水切り 取出指令
      OR      M1072  ; RB 水切り 取付指令
      OR      M1073  ; RB 後工程 右取付指令
      OR      M1074  ; RB 後工程 左取付指令
      OR      M1075  ; RB NG排出指令
      OR      M1076  ; RB 原点移動
      PLS     M911  ; RB Pro.ｽﾀｰﾄ
3322  LD      M911  ; RB Pro.ｽﾀｰﾄ
      OR      M912  ; RB Pro.ｽﾀｰﾄ 確認
      MPS
      ANI     T224  ; RB Pro.ｽﾀｰﾄ 遅延
      OUT     M912  ; RB Pro.ｽﾀｰﾄ 確認
      MPP
      OUT     T222 K3  ; RB Pro.ｽﾀｰﾄ 遅延
      MPS
      AND     T222  ; RB Pro.ｽﾀｰﾄ 遅延
      OUT     T223 K3  ; RB Pro.ｽﾀｰﾄ 遅延
      MPP
      AND     T223  ; RB Pro.ｽﾀｰﾄ 遅延
      OUT     T224 K10  ; RB Pro.ｽﾀｰﾄ 遅延
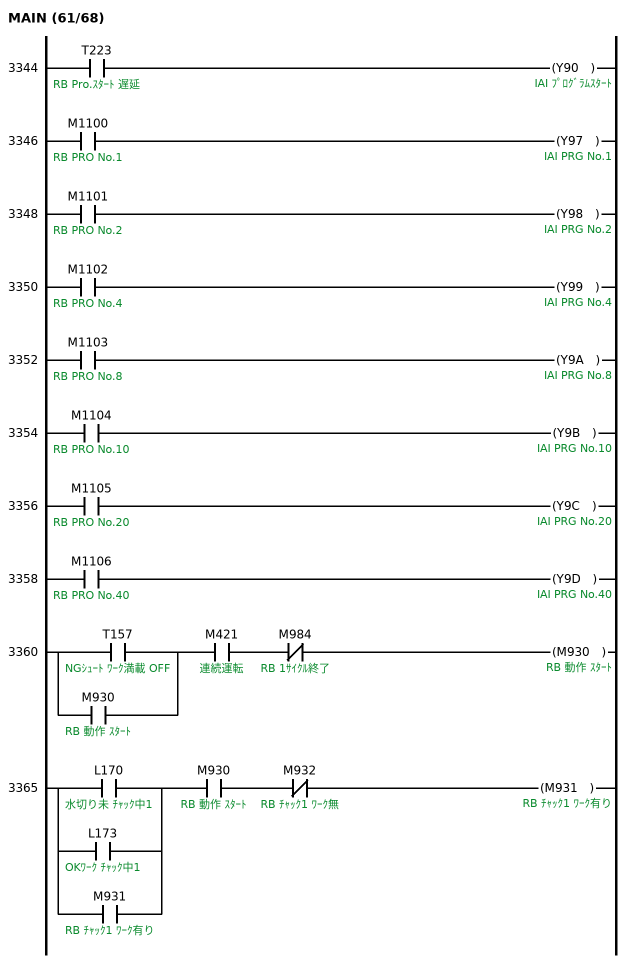
3344  LD      T223  ; RB Pro.ｽﾀｰﾄ 遅延
      OUT     Y90  ; IAI ﾌﾟﾛｸﾞﾗﾑｽﾀｰﾄ
3346  LD      M1100  ; RB PRO No.1
      OUT     Y97  ; IAI PRG No.1
3348  LD      M1101  ; RB PRO No.2
      OUT     Y98  ; IAI PRG No.2
3350  LD      M1102  ; RB PRO No.4
      OUT     Y99  ; IAI PRG No.4
3352  LD      M1103  ; RB PRO No.8
      OUT     Y9A  ; IAI PRG No.8
3354  LD      M1104  ; RB PRO No.10
      OUT     Y9B  ; IAI PRG No.10
3356  LD      M1105  ; RB PRO No.20
      OUT     Y9C  ; IAI PRG No.20
3358  LD      M1106  ; RB PRO No.40
      OUT     Y9D  ; IAI PRG No.40
3360  LD      T157  ; NGｼｭｰﾄ ﾜｰｸ満載 OFF
      OR      M930  ; RB 動作 ｽﾀｰﾄ
      AND     M421  ; 連続運転
      ANI     M984  ; RB 1ｻｲｸﾙ終了
      OUT     M930  ; RB 動作 ｽﾀｰﾄ
3365  LD      L170  ; 水切り未 ﾁｬｯｸ中1
      OR      L173  ; OKﾜｰｸ ﾁｬｯｸ中1
      OR      M931  ; RB ﾁｬｯｸ1 ﾜｰｸ有り
      AND     M930  ; RB 動作 ｽﾀｰﾄ
      ANI     M932  ; RB ﾁｬｯｸ1 ﾜｰｸ無
      OUT     M931  ; RB ﾁｬｯｸ1 ﾜｰｸ有り
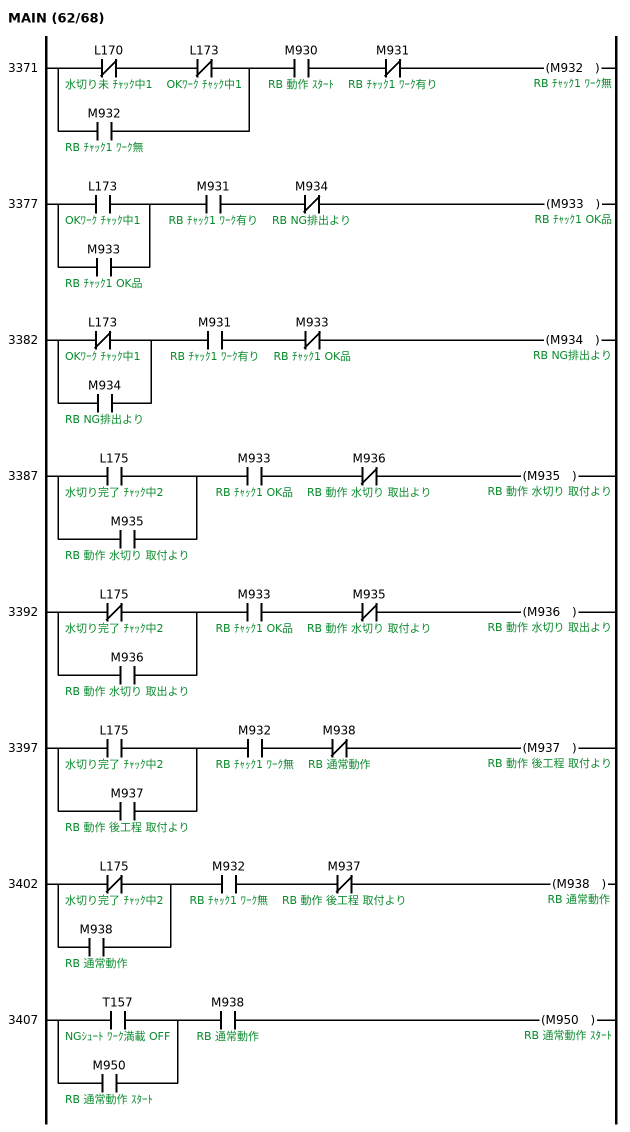
3371  LDI     L170  ; 水切り未 ﾁｬｯｸ中1
      ANI     L173  ; OKﾜｰｸ ﾁｬｯｸ中1
      OR      M932  ; RB ﾁｬｯｸ1 ﾜｰｸ無
      AND     M930  ; RB 動作 ｽﾀｰﾄ
      ANI     M931  ; RB ﾁｬｯｸ1 ﾜｰｸ有り
      OUT     M932  ; RB ﾁｬｯｸ1 ﾜｰｸ無
3377  LD      L173  ; OKﾜｰｸ ﾁｬｯｸ中1
      OR      M933  ; RB ﾁｬｯｸ1 OK品
      AND     M931  ; RB ﾁｬｯｸ1 ﾜｰｸ有り
      ANI     M934  ; RB NG排出より
      OUT     M933  ; RB ﾁｬｯｸ1 OK品
3382  LDI     L173  ; OKﾜｰｸ ﾁｬｯｸ中1
      OR      M934  ; RB NG排出より
      AND     M931  ; RB ﾁｬｯｸ1 ﾜｰｸ有り
      ANI     M933  ; RB ﾁｬｯｸ1 OK品
      OUT     M934  ; RB NG排出より
3387  LD      L175  ; 水切り完了 ﾁｬｯｸ中2
      OR      M935  ; RB 動作 水切り 取付より
      AND     M933  ; RB ﾁｬｯｸ1 OK品
      ANI     M936  ; RB 動作 水切り 取出より
      OUT     M935  ; RB 動作 水切り 取付より
3392  LDI     L175  ; 水切り完了 ﾁｬｯｸ中2
      OR      M936  ; RB 動作 水切り 取出より
      AND     M933  ; RB ﾁｬｯｸ1 OK品
      ANI     M935  ; RB 動作 水切り 取付より
      OUT     M936  ; RB 動作 水切り 取出より
3397  LD      L175  ; 水切り完了 ﾁｬｯｸ中2
      OR      M937  ; RB 動作 後工程 取付より
      AND     M932  ; RB ﾁｬｯｸ1 ﾜｰｸ無
      ANI     M938  ; RB 通常動作
      OUT     M937  ; RB 動作 後工程 取付より
3402  LDI     L175  ; 水切り完了 ﾁｬｯｸ中2
      OR      M938  ; RB 通常動作
      AND     M932  ; RB ﾁｬｯｸ1 ﾜｰｸ無
      ANI     M937  ; RB 動作 後工程 取付より
      OUT     M938  ; RB 通常動作
3407  LD      T157  ; NGｼｭｰﾄ ﾜｰｸ満載 OFF
      OR      M950  ; RB 通常動作 ｽﾀｰﾄ
      AND     M938  ; RB 通常動作
      OUT     M950  ; RB 通常動作 ｽﾀｰﾄ
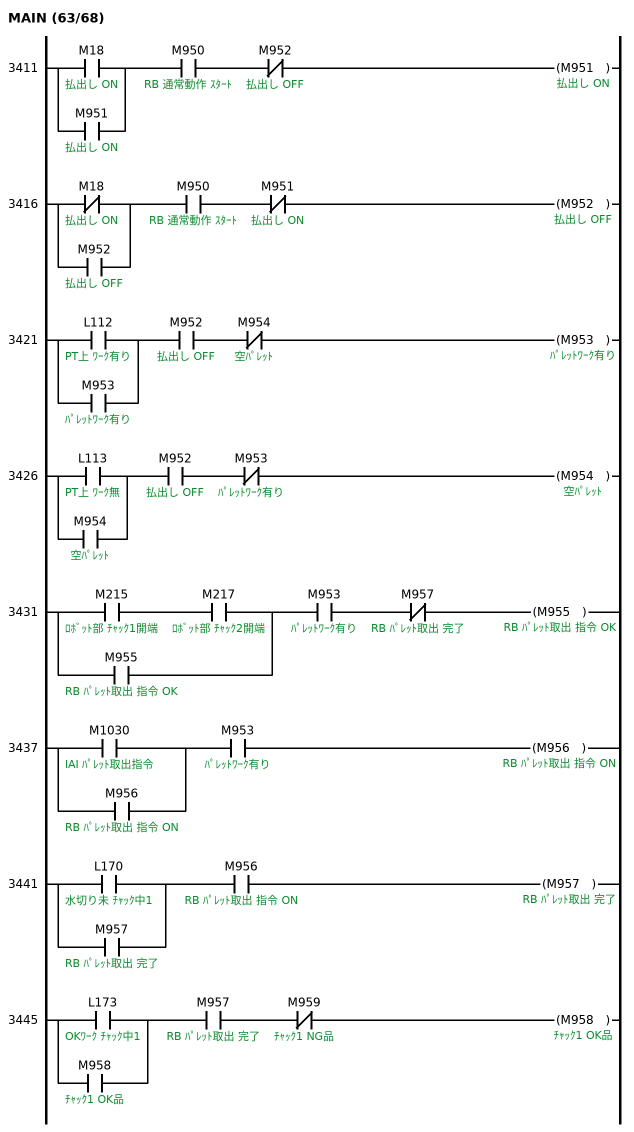
3411  LD      M18  ; 払出し ON
      OR      M951  ; 払出し ON
      AND     M950  ; RB 通常動作 ｽﾀｰﾄ
      ANI     M952  ; 払出し OFF
      OUT     M951  ; 払出し ON
3416  LDI     M18  ; 払出し ON
      OR      M952  ; 払出し OFF
      AND     M950  ; RB 通常動作 ｽﾀｰﾄ
      ANI     M951  ; 払出し ON
      OUT     M952  ; 払出し OFF
3421  LD      L112  ; PT上 ﾜｰｸ有り
      OR      M953  ; ﾊﾟﾚｯﾄﾜｰｸ有り
      AND     M952  ; 払出し OFF
      ANI     M954  ; 空ﾊﾟﾚｯﾄ
      OUT     M953  ; ﾊﾟﾚｯﾄﾜｰｸ有り
3426  LD      L113  ; PT上 ﾜｰｸ無
      OR      M954  ; 空ﾊﾟﾚｯﾄ
      AND     M952  ; 払出し OFF
      ANI     M953  ; ﾊﾟﾚｯﾄﾜｰｸ有り
      OUT     M954  ; 空ﾊﾟﾚｯﾄ
3431  LD      M215  ; ﾛﾎﾞｯﾄ部 ﾁｬｯｸ1開端
      AND     M217  ; ﾛﾎﾞｯﾄ部 ﾁｬｯｸ2開端
      OR      M955  ; RB ﾊﾟﾚｯﾄ取出 指令 OK
      AND     M953  ; ﾊﾟﾚｯﾄﾜｰｸ有り
      ANI     M957  ; RB ﾊﾟﾚｯﾄ取出 完了
      OUT     M955  ; RB ﾊﾟﾚｯﾄ取出 指令 OK
3437  LD      M1030  ; IAI ﾊﾟﾚｯﾄ取出指令
      OR      M956  ; RB ﾊﾟﾚｯﾄ取出 指令 ON
      AND     M953  ; ﾊﾟﾚｯﾄﾜｰｸ有り
      OUT     M956  ; RB ﾊﾟﾚｯﾄ取出 指令 ON
3441  LD      L170  ; 水切り未 ﾁｬｯｸ中1
      OR      M957  ; RB ﾊﾟﾚｯﾄ取出 完了
      AND     M956  ; RB ﾊﾟﾚｯﾄ取出 指令 ON
      OUT     M957  ; RB ﾊﾟﾚｯﾄ取出 完了
3445  LD      L173  ; OKﾜｰｸ ﾁｬｯｸ中1
      OR      M958  ; ﾁｬｯｸ1 OK品
      AND     M957  ; RB ﾊﾟﾚｯﾄ取出 完了
      ANI     M959  ; ﾁｬｯｸ1 NG品
      OUT     M958  ; ﾁｬｯｸ1 OK品
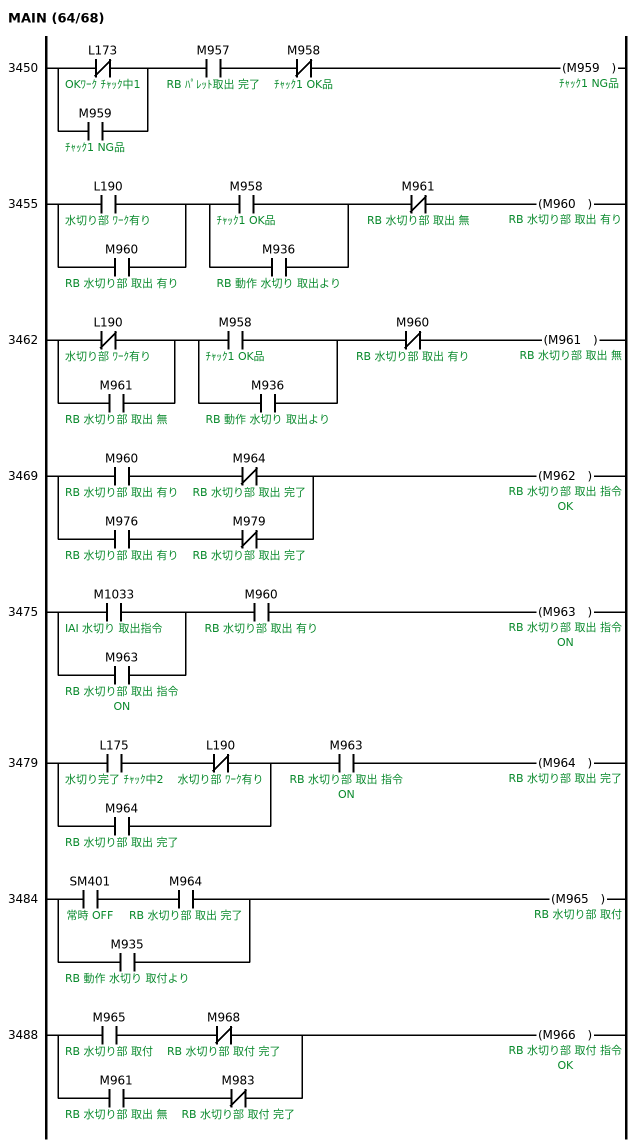
3450  LDI     L173  ; OKﾜｰｸ ﾁｬｯｸ中1
      OR      M959  ; ﾁｬｯｸ1 NG品
      AND     M957  ; RB ﾊﾟﾚｯﾄ取出 完了
      ANI     M958  ; ﾁｬｯｸ1 OK品
      OUT     M959  ; ﾁｬｯｸ1 NG品
3455  LD      L190  ; 水切り部 ﾜｰｸ有り
      OR      M960  ; RB 水切り部 取出 有り
      LD      M958  ; ﾁｬｯｸ1 OK品
      OR      M936  ; RB 動作 水切り 取出より
      ANB
      ANI     M961  ; RB 水切り部 取出 無
      OUT     M960  ; RB 水切り部 取出 有り
3462  LDI     L190  ; 水切り部 ﾜｰｸ有り
      OR      M961  ; RB 水切り部 取出 無
      LD      M958  ; ﾁｬｯｸ1 OK品
      OR      M936  ; RB 動作 水切り 取出より
      ANB
      ANI     M960  ; RB 水切り部 取出 有り
      OUT     M961  ; RB 水切り部 取出 無
3469  LD      M960  ; RB 水切り部 取出 有り
      ANI     M964  ; RB 水切り部 取出 完了
      LD      M976  ; RB 水切り部 取出 有り
      ANI     M979  ; RB 水切り部 取出 完了
      ORB
      OUT     M962  ; RB 水切り部 取出 指令 OK
3475  LD      M1033  ; IAI 水切り 取出指令
      OR      M963  ; RB 水切り部 取出 指令 ON
      AND     M960  ; RB 水切り部 取出 有り
      OUT     M963  ; RB 水切り部 取出 指令 ON
3479  LD      L175  ; 水切り完了 ﾁｬｯｸ中2
      ANI     L190  ; 水切り部 ﾜｰｸ有り
      OR      M964  ; RB 水切り部 取出 完了
      AND     M963  ; RB 水切り部 取出 指令 ON
      OUT     M964  ; RB 水切り部 取出 完了
3484  LD      SM401  ; 常時 OFF
      AND     M964  ; RB 水切り部 取出 完了
      OR      M935  ; RB 動作 水切り 取付より
      OUT     M965  ; RB 水切り部 取付
3488  LD      M965  ; RB 水切り部 取付
      ANI     M968  ; RB 水切り部 取付 完了
      LD      M961  ; RB 水切り部 取出 無
      ANI     M983  ; RB 水切り部 取付 完了
      ORB
      OUT     M966  ; RB 水切り部 取付 指令 OK
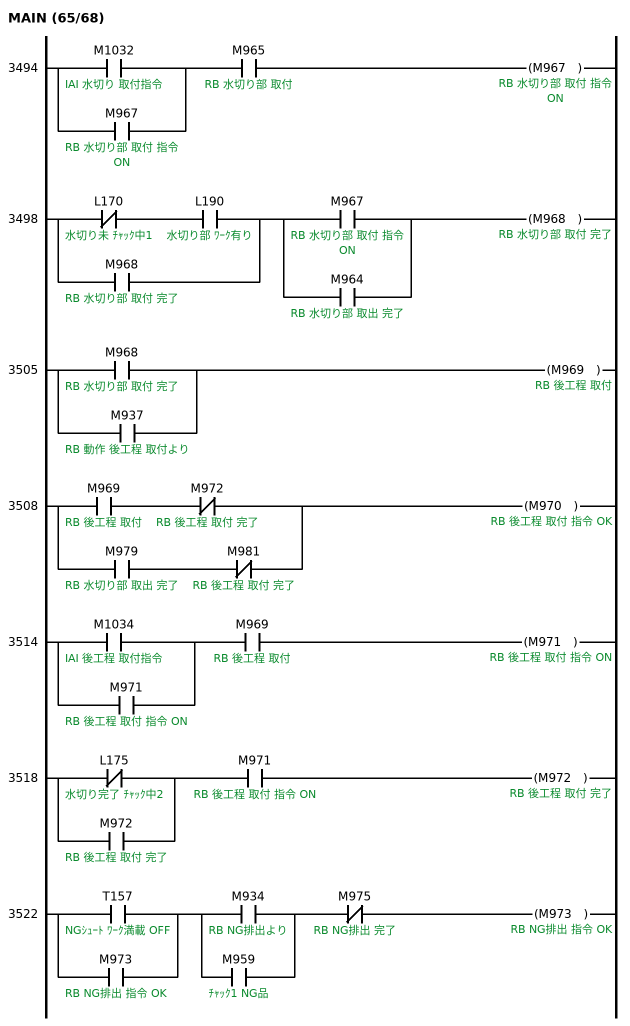
3494  LD      M1032  ; IAI 水切り 取付指令
      OR      M967  ; RB 水切り部 取付 指令 ON
      AND     M965  ; RB 水切り部 取付
      OUT     M967  ; RB 水切り部 取付 指令 ON
3498  LDI     L170  ; 水切り未 ﾁｬｯｸ中1
      AND     L190  ; 水切り部 ﾜｰｸ有り
      OR      M968  ; RB 水切り部 取付 完了
      LD      M967  ; RB 水切り部 取付 指令 ON
      OR      M964  ; RB 水切り部 取出 完了
      ANB
      OUT     M968  ; RB 水切り部 取付 完了
3505  LD      M968  ; RB 水切り部 取付 完了
      OR      M937  ; RB 動作 後工程 取付より
      OUT     M969  ; RB 後工程 取付
3508  LD      M969  ; RB 後工程 取付
      ANI     M972  ; RB 後工程 取付 完了
      LD      M979  ; RB 水切り部 取出 完了
      ANI     M981  ; RB 後工程 取付 完了
      ORB
      OUT     M970  ; RB 後工程 取付 指令 OK
3514  LD      M1034  ; IAI 後工程 取付指令
      OR      M971  ; RB 後工程 取付 指令 ON
      AND     M969  ; RB 後工程 取付
      OUT     M971  ; RB 後工程 取付 指令 ON
3518  LDI     L175  ; 水切り完了 ﾁｬｯｸ中2
      OR      M972  ; RB 後工程 取付 完了
      AND     M971  ; RB 後工程 取付 指令 ON
      OUT     M972  ; RB 後工程 取付 完了
3522  LD      T157  ; NGｼｭｰﾄ ﾜｰｸ満載 OFF
      OR      M973  ; RB NG排出 指令 OK
      LD      M934  ; RB NG排出より
      OR      M959  ; ﾁｬｯｸ1 NG品
      ANB
      ANI     M975  ; RB NG排出 完了
      OUT     M973  ; RB NG排出 指令 OK
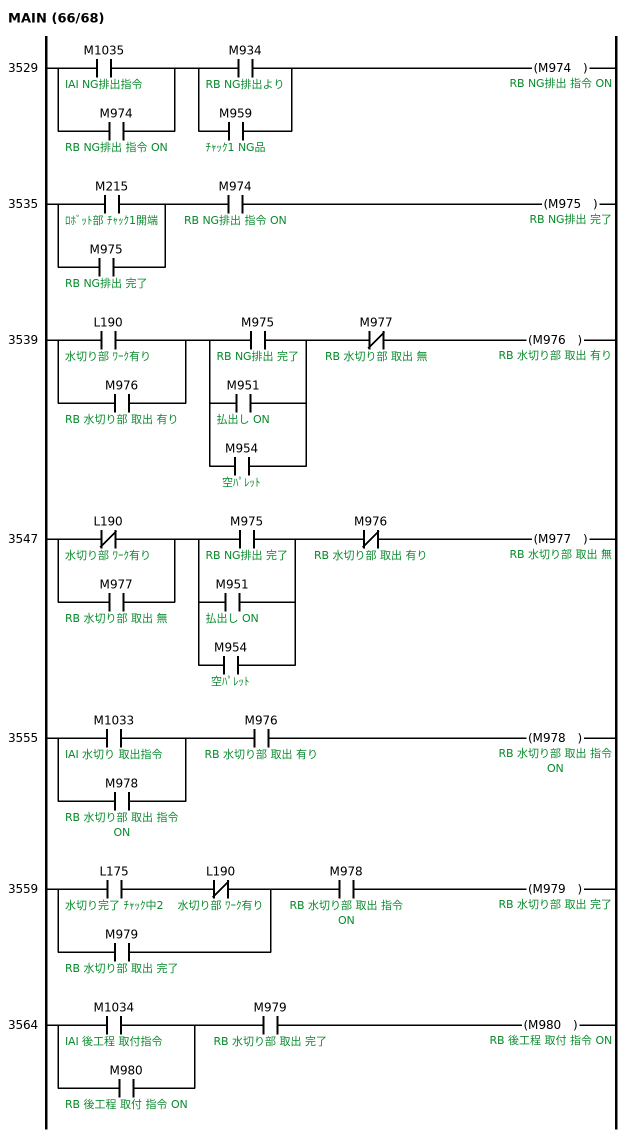
3529  LD      M1035  ; IAI NG排出指令
      OR      M974  ; RB NG排出 指令 ON
      LD      M934  ; RB NG排出より
      OR      M959  ; ﾁｬｯｸ1 NG品
      ANB
      OUT     M974  ; RB NG排出 指令 ON
3535  LD      M215  ; ﾛﾎﾞｯﾄ部 ﾁｬｯｸ1開端
      OR      M975  ; RB NG排出 完了
      AND     M974  ; RB NG排出 指令 ON
      OUT     M975  ; RB NG排出 完了
3539  LD      L190  ; 水切り部 ﾜｰｸ有り
      OR      M976  ; RB 水切り部 取出 有り
      LD      M975  ; RB NG排出 完了
      OR      M951  ; 払出し ON
      OR      M954  ; 空ﾊﾟﾚｯﾄ
      ANB
      ANI     M977  ; RB 水切り部 取出 無
      OUT     M976  ; RB 水切り部 取出 有り
3547  LDI     L190  ; 水切り部 ﾜｰｸ有り
      OR      M977  ; RB 水切り部 取出 無
      LD      M975  ; RB NG排出 完了
      OR      M951  ; 払出し ON
      OR      M954  ; 空ﾊﾟﾚｯﾄ
      ANB
      ANI     M976  ; RB 水切り部 取出 有り
      OUT     M977  ; RB 水切り部 取出 無
3555  LD      M1033  ; IAI 水切り 取出指令
      OR      M978  ; RB 水切り部 取出 指令 ON
      AND     M976  ; RB 水切り部 取出 有り
      OUT     M978  ; RB 水切り部 取出 指令 ON
3559  LD      L175  ; 水切り完了 ﾁｬｯｸ中2
      ANI     L190  ; 水切り部 ﾜｰｸ有り
      OR      M979  ; RB 水切り部 取出 完了
      AND     M978  ; RB 水切り部 取出 指令 ON
      OUT     M979  ; RB 水切り部 取出 完了
3564  LD      M1034  ; IAI 後工程 取付指令
      OR      M980  ; RB 後工程 取付 指令 ON
      AND     M979  ; RB 水切り部 取出 完了
      OUT     M980  ; RB 後工程 取付 指令 ON
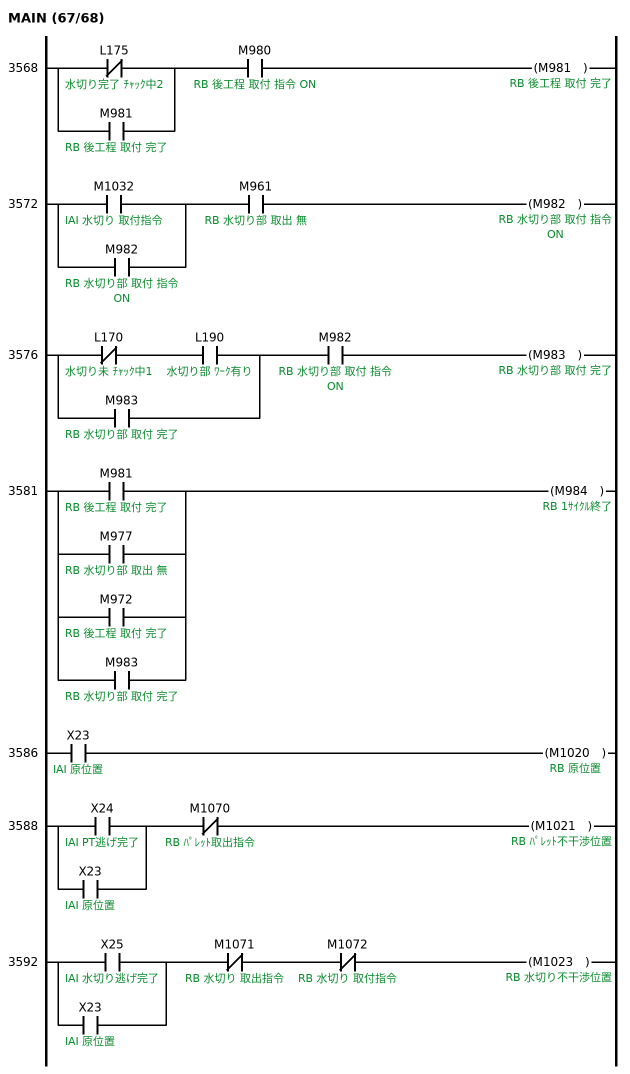
3568  LDI     L175  ; 水切り完了 ﾁｬｯｸ中2
      OR      M981  ; RB 後工程 取付 完了
      AND     M980  ; RB 後工程 取付 指令 ON
      OUT     M981  ; RB 後工程 取付 完了
3572  LD      M1032  ; IAI 水切り 取付指令
      OR      M982  ; RB 水切り部 取付 指令 ON
      AND     M961  ; RB 水切り部 取出 無
      OUT     M982  ; RB 水切り部 取付 指令 ON
3576  LDI     L170  ; 水切り未 ﾁｬｯｸ中1
      AND     L190  ; 水切り部 ﾜｰｸ有り
      OR      M983  ; RB 水切り部 取付 完了
      AND     M982  ; RB 水切り部 取付 指令 ON
      OUT     M983  ; RB 水切り部 取付 完了
3581  LD      M981  ; RB 後工程 取付 完了
      OR      M977  ; RB 水切り部 取出 無
      OR      M972  ; RB 後工程 取付 完了
      OR      M983  ; RB 水切り部 取付 完了
      OUT     M984  ; RB 1ｻｲｸﾙ終了
3586  LD      X23  ; IAI 原位置
      OUT     M1020  ; RB 原位置
3588  LD      X24  ; IAI PT逃げ完了
      OR      X23  ; IAI 原位置
      ANI     M1070  ; RB ﾊﾟﾚｯﾄ取出指令
      OUT     M1021  ; RB ﾊﾟﾚｯﾄ不干渉位置
3592  LD      X25  ; IAI 水切り逃げ完了
      OR      X23  ; IAI 原位置
      ANI     M1071  ; RB 水切り 取出指令
      ANI     M1072  ; RB 水切り 取付指令
      OUT     M1023  ; RB 水切り不干渉位置
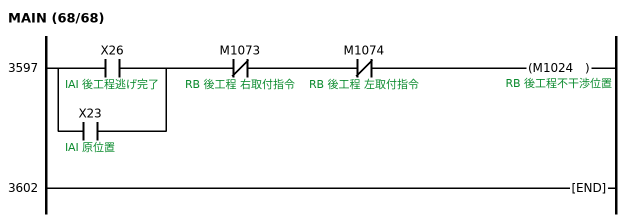
3597  LD      X26  ; IAI 後工程逃げ完了
      OR      X23  ; IAI 原位置
      ANI     M1073  ; RB 後工程 右取付指令
      ANI     M1074  ; RB 後工程 左取付指令
      OUT     M1024  ; RB 後工程不干渉位置
3602  END
END_PROGRAM

// device comments not shown above
M14  ; ﾌﾘｰﾌﾛｰ
M15  ; A-B制御
M20  ; 異常リセット
M21  ; PC電池異常
M22  ; ロボット電池異常
M23  ; プラグ異常
M24  ; エアー圧低下
M26  ; CC-LINK異常
M30  ; ﾜｰｸ押込みLS異常
M31  ; IDｾﾝｻｰ前後LS異常
M32  ; ﾜｰｸ押えLS異常
M33  ; ﾅｯﾄﾗﾝﾅｰ上下LS異常
M34  ; ﾊﾟﾚｯﾄ位置決めLS異常
M35  ; ﾅｯﾄﾗﾝﾅｰ部ｽﾄｯﾊﾟｰLS異常
M36  ; 水切りｼｬｯﾀｰLS異常
M37  ; ﾛﾎﾞｯﾄ部 ﾁｬｯｸ1 LS異常
M38  ; ﾛﾎﾞｯﾄ部 ﾁｬｯｸ2 LS異常
M39  ; 下降ﾘﾌﾀｰLS異常
M40  ; ｴｱｰﾌﾞﾛｰ部ｼｬｯﾀｰLS異常
M41  ; ｴｱｰﾌﾞﾛｰ部ｽﾄｯﾊﾟｰLS異常
M42  ; 旋回部旋回上下LS異常
M43  ; 旋回部旋回LS異常
M44  ; 押出し部ﾘﾌﾀｰLS異常
M45  ; 押出し部ﾌﾟｯｼｬｰLS異常
M46  ; ﾘﾀｰﾝ部ﾘﾌﾀｰLS異常
M47  ; ﾘﾀｰﾝ部ﾌﾟｯｼｬｰLS異常
M48  ; ロボット動作不可
M50  ; ﾛﾎﾞｯﾄCPU異常
M51  ; ﾛﾎﾞｯﾄ異常
M60  ; ﾅｯﾄﾗﾝﾅｰ前PT流動異常
M65  ; 出口部 PT流動異常
M66  ; 出口部 ｴｽｹｰﾌﾟ LS異常
M67  ; 出口部 ｽﾄｯﾊﾟｰ LS異常
M68  ; 搬入PT上下LS異常
M77  ; NGｼｭｰﾄ満載
M80  ; NGｼｭｰﾄLS異常
M96  ; NGパレット異常
M99  ; ID異常
M108  ; IAI運転中
M151  ; /ﾅｯﾄﾗﾝﾅｰ部異常補助
M163  ; MGｼｭｰﾄ部異常
M262  ; NGｼｭｰﾄ部原位置
M418  ; 洗浄搬送異常停止
M927  ; RB ﾁｬｯｸ1 完成品
M990  ; RB 水切り部 取付
M991  ; RB 水切り部 取付 有り
M992  ; RB 水切り部 取付 無
M993  ; RB 水切り部 取付 指令 OK
M994  ; RB 水切り部 取付 指令 ON
M995  ; RB 水切り部 取付 完了
M1000  ; RB ｶｺﾞ投入
M1001  ; RB ｶｺﾞ投入 有り
M1002  ; RB ｶｺﾞ投入 無
M1003  ; RB ｶｺﾞ投入 指令 OK
M1004  ; RB ｶｺﾞ投入 指令 ON
M1005  ; RB ｶｺﾞ投入 完了
M1009  ; RB 1ｻｲｸﾙ終了
M1051  ; 水切りモータ 速度 OK
M1053  ; 水切りモータ 回転数 OK
M1107  ; RB PRO No.80
M1900  ; ﾁｬｯｸ1 品番検索
M1901  ; 水切り 品番検索
M1902  ; ﾁｬｯｸ2 品番検索
M2000  ; 品番設定画面
M2001  ; 品番設定可
M2002  ; 設定品番書込み
M2010  ; 搬出指示データシフト
M2020  ; 生産指示画面
M2021  ; 生産指示書込み
M2031  ; 生産指示1書込み
M2032  ; 生産指示2書込み
M2033  ; 生産指示3書込み
M2034  ; 生産指示4書込み
M2035  ; 生産指示5書込み
M2036  ; 生産指示6書込み
M2041  ; 生産指示1消去
M2042  ; 生産指示2消去
M2043  ; 生産指示3消去
M2044  ; 生産指示4消去
M2045  ; 生産指示5消去
M2046  ; 生産指示6消去
M2050  ; 品番検索
M2051  ; 品番指示1番号検索
M2052  ; 品番指示2番号検索
M2053  ; 品番指示3番号検索
M2054  ; 品番指示4番号検索
M2055  ; 品番指示5番号検索
M2056  ; 品番指示6番号検索
M2100  ; ワークカウント
M2101  ; カウント一致あり
M2102  ; 新規カウント
M2500  ; ID条件
M2501  ; ID読み出し
M2502  ; TRG ON
M2503  ; TRG OFF
M2504  ; ID読み出し完了
M2510  ; ID書込み
M2511  ; TRG ON
M2512  ; TRG OFF
M2513  ; ID書込み完了
M2516  ; IDコマンド指令記憶
M2518  ; RESPONSE 1
M2520  ; TRG ON確認
L110  ; ID読込完了
L211  ; 第2搬送 工程完了
X1  ; ヒューズ正常
X2  ; エアー元圧正常
X5  ; ﾅｯﾄﾗﾝﾅｰ部搬送 INV異常
X6  ; 下降ﾘﾌﾀｰCV ｻｰﾏﾙﾄﾘｯﾌﾟ
X7  ; ｴｱｰﾌﾞﾛｰCV INV異常
X8  ; ﾘﾀｰﾝCV1 INV異常
X9  ; ﾘﾀｰﾝCV2 INV異常
X0E  ; 電磁ﾛｯｸ 閉
X20  ; IAI ｱﾗｰﾑ出力
X22  ; IAI 非常停止出力
X2C  ; IAI 汎用出力
X2D  ; IAI ｼｽﾃﾑﾒﾓﾘｰ ﾊﾞｯﾃﾘｰ警告
X2E  ; IAI ｱﾌﾞｿﾘｭｰﾄｴﾝｺｳﾀﾞｰ ﾊﾞｯﾃﾘｰ警告
X32  ; 第2搬送 搬送後退端
X36  ; 第2搬送 取出指令
X38  ; PT載せ換え工程 運転準備
X39  ; PT載せ換え工程 連続ﾓｰﾄﾞ
X3A  ; PT載せ換え工程 連続起動中
X40  ; 洗浄搬送装置 運転準備
X41  ; 洗浄搬送装置 扉閉め確認
X43  ; 洗浄搬送装置 搬送起動中
X50  ; ﾛﾎﾞｯﾄ ﾁｬｯｸ1閉端
X51  ; ﾛﾎﾞｯﾄ ﾁｬｯｸ1開端
X52  ; ﾛﾎﾞｯﾄ ﾁｬｯｸ2閉端
X53  ; ﾛﾎﾞｯﾄ ﾁｬｯｸ2開端
X54  ; PT載せ換え工程 運転準備
X55  ; 洗浄搬送装置 運転準備
X56  ; 洗浄搬送装置 扉閉め確認
X5E  ; 水切り ｼｬｯﾀｰ 開端
X5F  ; 水切り ｼｬｯﾀｰ 閉端
X110  ; READ DATA 0D0
X111  ; READ DATA 0D1
X112  ; READ DATA 0D2
X113  ; READ DATA 0D3
X114  ; READ DATA 0D4
X115  ; READ DATA 0D5
X116  ; READ DATA 0D6
X117  ; READ DATA 0D7
X118  ; NORMAL
X119  ; ERROR
X120  ; ユニット異常
X121  ; 自局ﾃﾞｰﾀﾘﾝｸ状態
X123  ; CC-LINK 異常局有
X126  ; CC-LINK ｽﾀｰﾄ　正常完了
X12F  ; ユニット レディ
X203  ; 異常リセットPB
X204  ; 教示入選択
X240  ; ﾜｰｸ押込み 前進端
X241  ; ﾜｰｸ押込み 後退端
X242  ; IDｾﾝｻｰ前後 前進端
X243  ; IDｾﾝｻｰ前後 後退端
X244  ; ﾜｰｸ押え 押え端
X245  ; ﾜｰｸ押え 戻し端
X247  ; ﾅｯﾄﾗﾝﾅｰ 下降端
X248  ; ﾊﾟﾚｯﾄ位置決め 端
X249  ; ﾊﾟﾚｯﾄ位置決め 戻し端
X24A  ; ﾊﾟﾚｯﾄｽﾄｯﾊﾟｰ 抜端
X24B  ; ﾊﾟﾚｯﾄｽﾄｯﾊﾟｰ 入端
X255  ; 下降ﾘﾌﾀｰ 下降端
X256  ; 下降ﾘﾌﾀｰ 上昇端
X257  ; 搬入PT上昇端
X258  ; 搬入PT下降端
X281  ; NGｼｭｰﾄ下降端
X282  ; ｴｱｰﾌﾞﾛｰ ｼｬｯﾀｰ 閉端
X283  ; ｴｱｰﾌﾞﾛｰ ｼｬｯﾀｰ 開端
X284  ; ｴｱｰﾌﾞﾛｰ ｽﾄｯﾊﾟｰ 抜き端
X285  ; ｴｱｰﾌﾞﾛｰ ｽﾄｯﾊﾟｰ 入り端
X286  ; 旋回上下 上昇端
X287  ; 旋回上下 下降端
X28A  ; 旋回部 旋回端
X28B  ; 旋回部 旋回戻し端
X28C  ; 押出し部 ﾌﾟｯｼｬｰ 前進端
X28D  ; 押出し部 ﾌﾟｯｼｬｰ 後退端
X291  ; ﾘﾀﾝｰ部 ﾘﾌﾀｰ上昇端
X292  ; ﾘﾀﾝｰ部 ﾘﾌﾀｰ下降端
X293  ; ﾘﾀｰﾝ部 ﾌﾟｯｼｬｰ 前進端
X294  ; ﾘﾀｰﾝ部 ﾌﾟｯｼｬｰ 後退端
X296  ; 押出し部 ﾘﾌﾀｰ上昇端
X297  ; 押出し部 ﾘﾌﾀｰ下降端
X298  ; 出口部 ｴｽｹｰﾌﾟ 入端
X299  ; 出口部 ｴｽｹｰﾌﾟ 抜端
X29A  ; 出口部 ｽﾄｯﾊﾟｰ 抜端
X29B  ; 出口部 ｽﾄｯﾊﾟｰ 入端
X29E  ; ルブリケータ下限
X1000  ; カウンタオールリセット
X1004  ; ID使用有 PB
X1005  ; ID使用無 PB
X1006  ; 工程No.有 PB
X1007  ; 工程No.無 PB
X1011  ; 品番設定SW
X1050  ; カウントリセット1
X1051  ; カウントリセット2
X1052  ; カウントリセット3
X1053  ; カウントリセット4
X1054  ; カウントリセット5
X1055  ; カウントリセット6
X1056  ; カウントリセット7
X1057  ; カウントリセット8
X1058  ; カウントリセット9
X1059  ; カウントリセット10
X105A  ; カウントリセット11
X1103  ; 水切ﾓｰﾀ停止 PB
X1111  ; ﾜｰｸ押込み 前進 PB
X1112  ; IDｾﾝｻｰ前後 後退 PB
X1113  ; IDｾﾝｻｰ前後 前進 PB
X1114  ; ﾊﾟﾚｯﾄｽﾄｯﾊﾟｰ 入 PB
X1115  ; ﾊﾟﾚｯﾄｽﾄｯﾊﾟｰ 抜 PB
X1116  ; ﾅｯﾄﾗﾝﾅｰ 下降 PB
X1117  ; ﾅｯﾄﾗﾝﾅｰ 上昇 PB
X1118  ; ﾊﾟﾚｯﾄ位置決め 戻し PB
X1119  ; ﾊﾟﾚｯﾄ位置決め  PB
X111A  ; ﾜｰｸ押え 戻し PB
X111B  ; ﾜｰｸ押え 押え PB
X111C  ; ﾅｯﾄﾗﾝﾅｰCV運転 PB
X111D  ; ﾅｯﾄﾗﾝﾅｰ運転 PB
X111E  ; 搬入PT上昇 PB
X111F  ; 搬入PT下降 PB
X1121  ; 下降ﾘﾌﾀｰ部 ﾘﾌﾀｰ上昇 PB
X1122  ; 下降ﾘﾌﾀｰ部 C/V搬入 PB
X1123  ; 下降ﾘﾌﾀｰ部 C/V搬出 PB
X1131  ; ﾛﾎﾞｯﾄ部 ﾁｬｯｸ1閉 PB
X1132  ; ﾛﾎﾞｯﾄ部 ﾁｬｯｸ2開 PB
X1133  ; ﾛﾎﾞｯﾄ部 ﾁｬｯｸ2閉 PB
X1134  ; ﾛﾎﾞｯﾄ原点復帰
X1141  ; 水切部 ｼｬｯﾀｰ閉 PB
X1142  ; 水切ﾓｰﾀ運転 PB
X1143  ; 水切ﾓｰﾀ原点復帰 PB
X1151  ; ｴｱｰﾌﾞﾛｰ ｼｬｯﾀｰ 閉 PB
X1152  ; ｴｱｰﾌﾞﾛｰ ｽﾄｯﾊﾟｰ 抜 PB
X1153  ; ｴｱｰﾌﾞﾛｰ ｽﾄｯﾊﾟｰ 入 PB
X1154  ; ｴｱｰﾌﾞﾛｰ入 PB
X1155  ; ｴｱｰﾌﾞﾛｰCV運転 PB
X1156  ; 旋回上下 下降 PB
X1157  ; 旋回上下 上昇 PB
X1158  ; 旋回部 旋回戻し PB
X1159  ; 旋回部 旋回 PB
X1161  ; 押出し部 ﾘﾌﾀｰ上昇PB
X1162  ; 押出し部 ﾌﾟｯｼｬｰ後退PB
X1163  ; 押出し部 ﾌﾟｯｼｬｰ前進PB
X1164  ; ﾘﾀｰﾝ部 ﾘﾌﾀｰ下降PB
X1165  ; ﾘﾀｰﾝ部 ﾘﾌﾀｰ上昇PB
X1166  ; ﾘﾀｰﾝ部 ﾌﾟｯｼｬｰ後退PB
X1167  ; ﾘﾀｰﾝ部 ﾌﾟｯｼｬｰ前進PB
X1168  ; ﾘﾀｰﾝC/V運転　PB
X1169  ; 出口部 ｴｽｹｰﾌﾟ抜 PB
X116A  ; 出口部 ｴｽｹｰﾌﾟ入 PB
X116B  ; 出口部 ｽﾄｯﾊﾟｰ入 PB
X116C  ; 出口部 ｽﾄｯﾊﾟｰ抜 PB
X11E1  ; ID書込み PB
X11E2  ; IDｾﾝｻｰ前後 後退 PB
X11E3  ; IDｾﾝｻｰ前後 前進 PB
X11EA  ; ID書込PB1
X11EB  ; ID書込データPB2
X11F0  ; ID書込ﾃﾞｰﾀ1
X11F1  ; ID書込ﾃﾞｰﾀ2
X1200  ; 設定品番書込み
X1480  ; 水切りモータ 速度 選択
X1482  ; 水切りモータ 回転数 選択
Y79  ; 洗浄搬送装置 品番情報2
Y7A  ; 洗浄搬送装置 品番情報4
Y7B  ; 洗浄搬送装置 品番情報8
Y7C  ; 洗浄搬送装置 品番情報10
Y7D  ; 洗浄搬送装置 品番情報20
Y7E  ; 洗浄搬送装置 品番情報40
Y7F  ; 洗浄搬送装置 品番情報80
Y95  ; IAI 一時停止解除
Y96  ; IAI 一時停止
Y0E4  ; 水切りﾓｰﾀｰ 実行禁止要求
Y120  ; WRITE DATA ID0
Y121  ; WRITE DATA ID1
Y122  ; WRITE DATA ID2
Y123  ; WRITE DATA ID3
Y124  ; WRITE DATA ID4
Y125  ; WRITE DATA ID5
Y126  ; WRITE DATA ID6
Y127  ; WRITE DATA ID7
Y128  ; R/W
Y129  ; INHIBIT/TRG
Y1004  ; ID使用有 PL
Y1005  ; ID使用無 PL
Y1006  ; 工程番号使用 PL
Y1007  ; 工程番号無し
Y1100  ; ﾅｯﾄﾗﾝﾅｰCV停止 PL
Y1101  ; ﾅｯﾄﾗﾝﾅｰ停止 PL
Y1102  ; 下降ﾘﾌﾀｰC/V停止 PL
Y1103  ; 水切ﾓｰﾀ停止 PL
Y1104  ; ｴｱｰﾌﾞﾛｰ停止 PL
Y1105  ; ｴｱｰﾌﾞﾛｰCV停止 PL
Y1106  ; ﾘﾀｰﾝC/V停止　PL
Y11E1  ; ID書込み 選択PL
Y11EA  ; ID書込データ1
Y11EB  ; ID書込データ2
Y11F0  ; ID書込ﾃﾞｰﾀ1
Y11F1  ; ID書込ﾃﾞｰﾀ2
Y1200  ; 設定品番書込み PL
Y1201  ; M10 PL
Y1202  ; M12 PL
Y1400  ; ﾅｯﾄﾗﾝﾅｰ部 原位置 PL
Y1401  ; 下降ﾘﾌﾀｰ部 原位置 PL
Y1402  ; ﾛﾎﾞｯﾄ部 原位置 PL
Y1403  ; 水切部 原位置 PL
Y1404  ; ｴｱｰﾌﾞﾛｰ部&旋回部 原位置 PL
Y1405  ; ﾘﾀｰﾝ部 原位置 PL
Y1410  ; ﾜｰｸ押込み 後退 端PL
Y1411  ; ﾜｰｸ押込み 前進 端PL
Y1412  ; IDｾﾝｻｰ前後 後退 端PL
Y1413  ; IDｾﾝｻｰ前後 前進 端PL
Y1414  ; ﾊﾟﾚｯﾄｽﾄｯﾊﾟｰ 入 端PL
Y1415  ; ﾊﾟﾚｯﾄｽﾄｯﾊﾟｰ 抜 端PL
Y1416  ; ﾅｯﾄﾗﾝﾅｰ 下降 端PL
Y1417  ; ﾅｯﾄﾗﾝﾅｰ 上昇 端PL
Y1418  ; ﾊﾟﾚｯﾄ位置決め 戻し 端PL
Y1419  ; ﾊﾟﾚｯﾄ位置決め  端PL
Y141A  ; ﾜｰｸ押え 戻し 端PL
Y141B  ; ﾜｰｸ押え 押え 端PL
Y141C  ; ﾅｯﾄﾗﾝﾅｰCV運転 PL
Y141D  ; ﾅｯﾄﾗﾝﾅｰ運転 PL
Y141E  ; 搬入PT上昇 端PL
Y141F  ; 搬入PT下降 端PL
Y1420  ; 下降ﾘﾌﾀｰ部 ﾘﾌﾀｰ下降 端PL
Y1421  ; 下降ﾘﾌﾀｰ部 ﾘﾌﾀｰ上昇 端PL
Y1422  ; 下降ﾘﾌﾀｰ部 C/V搬入 PL
Y1423  ; 下降ﾘﾌﾀｰ部 C/V搬出 PL
Y1430  ; ﾛﾎﾞｯﾄ部 ﾁｬｯｸ1開 端PL
Y1431  ; ﾛﾎﾞｯﾄ部 ﾁｬｯｸ1閉 端PL
Y1432  ; ﾛﾎﾞｯﾄ部 ﾁｬｯｸ2開 端PL
Y1433  ; ﾛﾎﾞｯﾄ部 ﾁｬｯｸ2閉 端PL
Y1434  ; ﾛﾎﾞｯﾄ原点復帰 PL
Y1440  ; 水切部 ｼｬｯﾀｰ開 端PL
Y1441  ; 水切部 ｼｬｯﾀｰ閉 端PL
Y1442  ; 水切ﾓｰﾀ運転 端PL
Y1443  ; 水切ﾓｰﾀ原点復帰 PL
Y1450  ; ｴｱｰﾌﾞﾛｰ ｼｬｯﾀｰ 開 端PL
Y1451  ; ｴｱｰﾌﾞﾛｰ ｼｬｯﾀｰ 閉 端PL
Y1452  ; ｴｱｰﾌﾞﾛｰ ｽﾄｯﾊﾟｰ 抜 端PL
Y1453  ; ｴｱｰﾌﾞﾛｰ ｽﾄｯﾊﾟｰ 入 端PL
Y1454  ; ｴｱｰﾌﾞﾛｰ入 PL
Y1455  ; ｴｱｰﾌﾞﾛｰCV運転 PL
Y1456  ; 旋回上下 下降 端PL
Y1457  ; 旋回上下 上昇 端PL
Y1458  ; 旋回部 旋回戻し 端PL
Y1459  ; 旋回部 旋回 端PL
Y1460  ; 押出し部 ﾘﾌﾀｰ下降端 PL
Y1461  ; 押出し部 ﾘﾌﾀｰ上昇端 PL
Y1462  ; 押出し部 ﾌﾟｯｼｬｰ後退端 PL
Y1463  ; 押出し部 ﾌﾟｯｼｬｰ前進端 PL
Y1464  ; ﾘﾀｰﾝ部 ﾘﾌﾀｰ下降端 PL
Y1465  ; ﾘﾀｰﾝ部 ﾘﾌﾀｰ上昇端 PL
Y1466  ; ﾘﾀｰﾝ部 ﾌﾟｯｼｬｰ後退端 PL
Y1467  ; ﾘﾀｰﾝ部 ﾌﾟｯｼｬｰ前進端 PL
Y1468  ; ﾘﾀｰﾝC/V運転　PL
Y1469  ; 出口部 ｴｽｹｰﾌﾟ抜 端PL
Y146A  ; 出口部 ｴｽｹｰﾌﾟ入 端PL
Y146B  ; 出口部 ｽﾄｯﾊﾟｰ入 端PL
Y146C  ; 出口部 ｽﾄｯﾊﾟｰ抜 端PL
Y1480  ; 水切りモータ 速度 選択
Y1482  ; 水切りモータ 回転数 選択
Y14E0  ; ID読出し PL
Y14E1  ; ID書込み PL
Y14E2  ; IDｾﾝｻｰ前後 後退 端PL
Y14E3  ; IDｾﾝｻｰ前後 前進 端PL
Y14EF  ; ID異常 PL
Y1500  ; カウント表示
Y1501  ; 気圧
Y1502  ; 運転準備
Y1503  ; 各個
Y1504  ; 連続
Y1505  ; 教示
Y1506  ; 原位置
Y1507  ; ｻｲｸﾙ中
Y150A  ; ｻｰﾎﾞON
Y150B  ; ﾌﾟﾗｸﾞOK
Y150C  ; 教示可
Y1510  ; 品番設定可
B1  ; PC電池異常
B2  ; ロボット電池異常
B3  ; プラグ異常
B4  ; エアー圧低下
B5  ; サーボ異常
B6  ; CC-LINK異常
B0A  ; ﾜｰｸ押込みLS異常
B0B  ; IDｾﾝｻｰ前後LS異常
B0C  ; ﾜｰｸ押えLS異常
B0D  ; ﾅｯﾄﾗﾝﾅｰ上下LS異常
B0E  ; ﾊﾟﾚｯﾄ位置決めLS異常
B0F  ; ﾅｯﾄﾗﾝﾅｰ部ｽﾄｯﾊﾟｰLS異常
B10  ; 水切りｼｬｯﾀｰLS異常
B11  ; ﾛﾎﾞｯﾄ部 ﾁｬｯｸ1 LS異常
B12  ; ﾛﾎﾞｯﾄ部 ﾁｬｯｸ2 LS異常
B13  ; 下降ﾘﾌﾀｰLS異常
B14  ; ｴｱｰﾌﾞﾛｰ部ｼｬｯﾀｰLS異常
B15  ; ｴｱｰﾌﾞﾛｰ部ｽﾄｯﾊﾟｰLS異常
B16  ; 旋回部旋回上下LS異常
B17  ; 旋回部旋回LS異常
B18  ; 押出し部ﾘﾌﾀｰLS異常
B19  ; 押出し部ﾌﾟｯｼｬｰLS異常
B1A  ; ﾘﾀｰﾝ部ﾘﾌﾀｰLS異常
B1B  ; ﾘﾀｰﾝ部ﾌﾟｯｼｬｰLS異常
B1C  ; ロボット動作不可
B1E  ; ﾛﾎﾞｯﾄCPU異常
B1F  ; ﾛﾎﾞｯﾄ異常
B20  ; ﾅｯﾄﾗﾝﾅｰ部搬送CV INV異常
B21  ; 下降ﾘﾌﾀｰCV ｻｰﾏﾙﾄﾘｯﾌﾟ
B22  ; ｴｱｰﾌﾞﾛｰ部搬送CV INV異常
B23  ; ﾘﾀｰﾝCV INV異常
B32  ; ｴｱｰﾓｰﾀｰ ﾎﾞﾙﾄ緩め異常
B39  ; NGｼｭｰﾄ満載
B40  ; 出口部 ｴｽｹｰﾌﾟ 動作異常
B41  ; 出口部 ｽﾄｯﾊﾟｰ 動作異常
B42  ; NGパレット異常
B45  ; ID異常
B46  ; ﾜｰｸ押込み動作異常
B47  ; IDｾﾝｻｰ前後動作異常
B48  ; ﾜｰｸ押え動作異常
B49  ; ﾅｯﾄﾗﾝﾅｰ上下動作異常
B4A  ; ﾊﾟﾚｯﾄ位置決め動作異常
B4B  ; ﾅｯﾄﾗﾝﾅｰ部ｽﾄｯﾊﾟｰ動作異常
B4C  ; 水切りｼｬｯﾀｰ動作異常
B4D  ; ﾛﾎﾞｯﾄ部ﾁｬｯｸ1動作異常
B4E  ; ﾛﾎﾞｯﾄ部ﾁｬｯｸ2動作異常
B4F  ; 下降ﾘﾌﾀｰ動作異常
B50  ; ｴｱｰﾌﾞﾛｰ部ｼｬｯﾀｰ動作異常
B51  ; ｴｱｰﾌﾞﾛｰ部ｽﾄｯﾊﾟｰ動作異常
B52  ; 旋回部旋回上下動作異常
B53  ; 旋回部旋回動作異常
B54  ; 押出し部ﾘﾌﾀｰ動作異常
B55  ; 押出し部ﾌﾟｯｼｬｰ動作異常
B56  ; ﾘﾀｰﾝ部ﾘﾌﾀｰ動作異常
B57  ; ﾘﾀｰﾝ部ﾌﾟｯｼｬｰ動作異常
B58  ; 搬入PT上下 動作異常
B59  ; 自動 ﾘﾀｰﾝCV停止
D8  ; 画面切り替え
D811  ; RB ﾁｬﾂｸ1 品番
D812  ; 水切り部 品番
D813  ; RB ﾁｬｯｸ2 品番
D821  ; RB ﾁｬﾂｸ1 ﾜｰｸ種類
D822  ; 水切り部 ﾜｰｸ種類
D823  ; RB ﾁｬｯｸ2 ﾜｰｸ種類
D900  ; 軸1 ERROR CODE
D930  ; 水切りモータ 速度 画面
D931  ; 水切りモータ 回転数 画面
D950  ; 水切りモータ 速度
D951  ; 水切りモータ 速度
D952  ; 水切りモータ 回転数
D953  ; 水切りモータ 回転数
D1000  ; 水切り 単位設定
D1001  ; 水切り 単位倍率
D1002  ; 水切り 1回転ﾊﾟﾙｽ数
D1003  ; 水切り 1回転ﾊﾟﾙｽ数
D1004  ; 水切り 1回転移動量
D1005  ; 水切り 1回転移動量
D1008  ; 水切り ﾊﾞｲｱｽ速度
D1009  ; 水切り ﾊﾞｲｱｽ速度
D1010  ; 水切り 速度制限値
D1011  ; 水切り 速度制限値
D1012  ; 水切り 加速時間
D1013  ; 水切り 加速時間
D1014  ; 水切り 減速時間
D1015  ; 水切り 減速時間
D1017  ; 水切り ﾊﾞｯｸﾗｯｼｭ補正量
D1018  ; 水切り ｿﾌﾄﾘﾐｯﾄ上限値
D1019  ; 水切り ｿﾌﾄﾘﾐｯﾄ上限値
D1020  ; 水切り ｿﾌﾄﾘﾐｯﾄ下限値
D1021  ; 水切り ｿﾌﾄﾘﾐｯﾄ下限値
D1022  ; 水切り ｿﾌﾄﾘﾐｯﾄ選択
D1023  ; 水切り ｿﾌﾄﾘﾐｯﾄ有効
D1024  ; 水切り 指令ｲﾝﾎﾟｼﾞｼｮﾝ範囲
D1025  ; 水切り 指令ｲﾝﾎﾟｼﾞｼｮﾝ範囲
D1026  ; 水切り ﾄﾙｸ制限設定値
D1027  ; 水切り Mｺｰﾄﾞ出力ﾀｲﾐﾝｸﾞ
D1028  ; 水切り 速度切替ﾓｰﾄﾞ
D1029  ; 水切り 補間速度指定方法
D1030  ; 水切り 速度制御時の送り現在値
D1031  ; 水切り 入力信号論理選択
D1033  ; 水切り 手動ﾊﾟﾙｻ入力選択
D1034  ; 水切り 速度・位置機能選択
D1036  ; 水切り 加速時間１
D1037  ; 水切り 加速時間１
D1038  ; 水切り 加速時間２
D1039  ; 水切り 加速時間２
D1040  ; 水切り 加速時間３
D1041  ; 水切り 加速時間３
D1042  ; 水切り 減速時間１
D1043  ; 水切り 減速時間１
D1044  ; 水切り 減速時間２
D1045  ; 水切り 減速時間２
D1046  ; 水切り 減速時間３
D1047  ; 水切り 減速時間３
D1048  ; 水切り JOG速度制限値
D1049  ; 水切り JOG速度制限値
D1050  ; 水切り JOG運転加速時間選択
D1051  ; 水切り JOG運転減速時間選択
D1052  ; 水切り 加減速処理選択
D1053  ; 水切り S字比率
D1054  ; 水切り 急停止減速時間
D1055  ; 水切り 急停止減速時間
D1056  ; 水切り 停止ｸﾞﾙｰﾌﾟ1急停止選択
D1057  ; 水切り 停止ｸﾞﾙｰﾌﾟ2急停止選択
D1058  ; 水切り 停止ｸﾞﾙｰﾌﾟ3急停止選択
D1059  ; 水切り 位置決め完了信号出力時間
D1060  ; 水切り 円弧補間誤差許容範囲
D1061  ; 水切り 円弧補間誤差許容範囲
D1062  ; 水切り 外部指令機能選択
D1064  ; 水切り 再始動許容範囲設定
D1065  ; 水切り 再始動許容範囲設定
D1070  ; 水切り 原点復帰方式
D1071  ; 水切り 原点復帰方向
D1072  ; 水切り 原点ｱﾄﾞﾚｽ
D1073  ; 水切り 原点ｱﾄﾞﾚｽ
D1074  ; 水切り 原点復帰速度
D1075  ; 水切り 原点復帰速度
D1076  ; 水切り ｸﾘｰﾌﾟ速度
D1077  ; 水切り ｸﾘｰﾌﾟ速度
D1078  ; 水切り 原点復帰ﾘﾄﾗｲ
D1100  ; 水切り ｻｰﾎﾞｼﾘｰｽﾞ
D1101  ; 水切り ｱﾝﾌﾟ設定
D1102  ; 水切り 回生抵抗
D1103  ; 水切り ﾓｰﾀﾀｲﾌﾟ
D1104  ; 水切り ﾓｰﾀ容量
D1105  ; 水切り ﾓｰﾀ回転数
D1106  ; 水切り ﾌｨｰﾄﾞﾊﾞｯｸﾊﾟﾙｽ
D1107  ; 水切り 回転方向
D1108  ; 水切り ｵｰﾄﾁｭｰﾆﾝｸﾞ
D1109  ; 水切り ｻｰﾎﾞ応答性設定
D1200  ; 水切り NO.1 位置決め識別子
D1201  ; 水切り NO.1 Mｺｰﾄﾞ
D1202  ; 水切り NO.1 ﾄﾞｩｴﾙﾀｲﾑ
D1204  ; 水切り NO.1 指令速度
D1206  ; 水切り NO.1 位置決めｱﾄﾞﾚｽ
D1210  ; 水切り NO.2 位置決め識別子
D1211  ; 水切り NO.2 Mｺｰﾄﾞ
D1212  ; 水切り NO.2 ﾄﾞｩｴﾙﾀｲﾑ
D1214  ; 水切り NO.2 指令速度
D1216  ; 水切り NO.2 位置決めｱﾄﾞﾚｽ
D7000  ; 品番検索結果
D7001  ; 品番一致数
D7002  ; 品番検索結果*2
T0  ; 電源入り確認1
T1  ; 電源入り確認2
T10  ; 集中警報切
T11  ; 集中警報入
T12  ; 着座無効
T13  ; 着座有効
T14  ; ﾌﾘｰﾌﾛｰ
T15  ; A-B制御
T16  ; 教示モード
T20  ; エアー元圧低下
T30  ; ﾜｰｸ押込み動作異常
T31  ; IDｾﾝｻｰ前後動作異常
T32  ; ﾜｰｸ押え動作異常
T33  ; ﾅｯﾄﾗﾝﾅｰ上下動作異常
T34  ; ﾊﾟﾚｯﾄ位置決め動作異常
T35  ; ﾅｯﾄﾗﾝﾅｰ部ｽﾄｯﾊﾟｰ動作異常
T36  ; 水切りｼｬｯﾀｰ動作異常
T37  ; ﾛﾎﾞｯﾄ部ﾁｬｯｸ1動作異常
T38  ; ﾛﾎﾞｯﾄ部ﾁｬｯｸ2動作異常
T39  ; 下降ﾘﾌﾀｰ動作異常
T40  ; ｴｱｰﾌﾞﾛｰ部ｼｬｯﾀｰ動作異常
T41  ; ｴｱｰﾌﾞﾛｰ部ｽﾄｯﾊﾟｰ動作異常
T42  ; 旋回部旋回上下動作異常
T43  ; 旋回部旋回動作異常
T44  ; 押出し部ﾘﾌﾀｰ動作異常
T45  ; 押出し部ﾌﾟｯｼｬｰ動作異常
T46  ; ﾘﾀｰﾝ部ﾘﾌﾀｰ動作異常
T47  ; ﾘﾀｰﾝ部ﾌﾟｯｼｬｰ動作異常
T50  ; 出口部 ｴｽｹｰﾌﾟ 動作異常
T51  ; 出口部 ｽﾄｯﾊﾟｰ 動作異常
T52  ; 搬入PT上下 動作異常
T53  ; NGｼｭｰﾄ動作異常
T60  ; ﾅｯﾄﾗﾝﾅｰ前PT流動異常
T65  ; 出口部 PT流動異常
T100  ; 空ｶｺﾞ減少
T108  ; ID読出しタイムオーバー
T109  ; ID書込みタイムオーバー
T220  ; ﾛﾎﾞｯﾄｻｰﾎﾞON指示
T221  ; ロボット異常ﾘｾｯﾄ指示
T228  ; カウント出力時間
T229  ; カウント表示時間
T230  ; ﾊﾞﾘ取り機へ自動起動指令 切り
T231  ; ﾊﾞﾘ取機へ 治具洗浄要求 切り
T250  ; ID読み出しTRG
T252  ; ID書込み TRG
T253  ; TRG ON確認
